// TIA Portal V20 program export: 1 tag tables, 2 data types, 6 data blocks, 9 code blocks (in call order from the OBs), 0 instance data blocks

VAR_GLOBAL   // PLC tag table "Default tag table"
   OpenCmd AT %M0.0 : Bool;
   CloseCmd AT %M0.1 : Bool;
   OpenFB AT %M0.2 : Bool;
   ClosedFB AT %M0.3 : Bool;
   LocalMode AT %M0.4 : Bool;
   Healthy AT %M0.5 : Bool;
   OpenValve AT %M0.6 : Bool;
   CloseValve AT %M0.7 : Bool;
   Tag__639217692550262421 AT %I2.0 : Bool;
   Tag__639217692553776870 AT %I2.1 : Bool;
   Tag__639217692553954872 AT %I2.2 : Bool;
   Tag__639217692553954873 AT %I2.3 : Bool;
   Tag__639217692554216438 AT %I2.4 : Bool;
   Tag__639217692554394622 AT %I2.5 : Bool;
   Tag__639217692554432300 AT %I2.6 : Bool;
   Tag__639217692556336031 AT %I2.7 : Bool;
   Tag__639217692556550149 AT %I3.0 : Bool;
   Tag__639217692556680608 AT %I3.1 : Bool;
   Tag__639217692556821735 AT %I3.2 : Bool;
   Tag__639217692556891742 AT %I3.3 : Bool;
   Tag__639217692557049682 AT %I3.4 : Bool;
   Tag__639217692557209508 AT %I3.5 : Bool;
   Tag__639217692557209509 AT %I3.6 : Bool;
   Tag__639217692557471753 AT %I3.7 : Bool;
   Tag__639217692557529414 AT %I4.0 : Bool;
   Tag__639217692557689863 AT %I4.1 : Bool;
   Tag__639217692557850060 AT %I4.2 : Bool;
   Tag__639217692558010331 AT %I4.3 : Bool;
   Tag__639217692558171799 AT %I4.4 : Bool;
   Tag__639217692558331401 AT %I4.5 : Bool;
   Tag__639217692558488410 AT %I4.6 : Bool;
   Tag__639217692558802162 AT %I4.7 : Bool;
   Tag__639217692558961456 AT %I5.0 : Bool;
   Tag__639217692558971616 AT %I5.1 : Bool;
   Tag__639217692559129482 AT %I5.2 : Bool;
   Tag__639217692559281543 AT %I5.3 : Bool;
   Tag__639217692559443162 AT %I5.4 : Bool;
   Tag__639217692559601745 AT %I5.5 : Bool;
   Tag__639217692559760896 AT %I5.6 : Bool;
   Tag__639217692559921432 AT %I5.7 : Bool;
   Tag__639217692559921433 AT %I6.0 : Bool;
   Tag__639217692560082018 AT %I6.1 : Bool;
   Tag__639217692560402934 AT %I6.2 : Bool;
   Tag__639217692560402935 AT %I6.3 : Bool;
   Tag__639217692560583987 AT %I6.4 : Bool;
   Tag__639217692560723706 AT %I6.5 : Bool;
   Tag__639217692560880740 AT %I6.6 : Bool;
   Tag__639217692561041807 AT %I6.7 : Bool;
   Tag__639217692561206457 AT %I7.0 : Bool;
   Tag__639217692561359218 AT %I7.1 : Bool;
   Tag__639217692561520184 AT %I7.2 : Bool;
   Tag__639217692561520185 AT %I7.3 : Bool;
   Tag__639217692561802187 AT %I7.4 : Bool;
   Tag__639217692561935087 AT %I7.5 : Bool;
   Tag__639217692562065024 AT %I7.6 : Bool;
   Tag__639217692562223286 AT %I7.7 : Bool;
   Tag__639217692562383723 AT %I8.0 : Bool;
   Tag__639217692562543936 AT %I8.1 : Bool;
   Tag__639217692562543937 AT %I8.2 : Bool;
   Tag__639217692562862407 AT %I8.3 : Bool;
   Tag__639217692562862408 AT %I8.4 : Bool;
   Tag__639217692563093001 AT %I8.5 : Bool;
   Tag__639217692563182212 AT %I8.6 : Bool;
   Tag__639217692563343596 AT %I8.7 : Bool;
   Tag__639217692563511187 AT %I9.0 : Bool;
   Tag__639217692563662093 AT %I9.1 : Bool;
   Tag__639217692563662094 AT %I9.2 : Bool;
   Tag__639217692563823907 AT %I9.3 : Bool;
   Tag__639217692566083593 AT %I9.4 : Bool;
   Tag__639217692566201557 AT %I9.5 : Bool;
   Tag__639217692566360040 AT %I9.6 : Bool;
   Tag__639217692566517145 AT %I9.7 : Bool;
   Tag__639217692566674032 AT %I10.0 : Bool;
   Tag__639217692566832496 AT %I10.1 : Bool;
   Tag__639217692566832497 AT %I10.2 : Bool;
   Tag__639217692567184922 AT %I10.3 : Bool;
   Tag__639217692567336780 AT %I10.4 : Bool;
   Tag__639217692567388945 AT %I10.5 : Bool;
   Tag__639217692567546587 AT %I10.6 : Bool;
   Tag__639217692567707146 AT %I10.7 : Bool;
   Tag__639217692567868007 AT %I11.0 : Bool;
   Tag__639217692567868008 AT %I11.1 : Bool;
   Tag__639217692568025035 AT %I11.2 : Bool;
   Tag__639217692568182907 AT %I11.3 : Bool;
   Tag__639217692568341074 AT %I11.4 : Bool;
   Tag__639217692568550097 AT %I11.5 : Bool;
   Tag__639217692568683019 AT %I11.6 : Bool;
   Tag__639217692568840948 AT %I11.7 : Bool;
   Tag__639217692568971320 AT %I12.0 : Bool;
   Tag__639217692569119475 AT %I12.1 : Bool;
   Tag__639217692569298523 AT %I12.2 : Bool;
   Tag__639217692569460008 AT %I12.3 : Bool;
   Tag__639217692569619373 AT %I12.4 : Bool;
   Tag__639217692569780777 AT %I12.5 : Bool;
   Tag__639217692569780778 AT %I12.6 : Bool;
   Tag__639217692569942097 AT %I12.7 : Bool;
   Tag__639217692570102018 AT %I13.0 : Bool;
   Tag__639217692570262026 AT %I13.1 : Bool;
   Tag__639217692570422186 AT %I13.2 : Bool;
   Tag__639217692570422187 AT %I13.3 : Bool;
   Tag__639217692570583489 AT %I13.4 : Bool;
   Tag__639217692570745102 AT %I13.5 : Bool;
   Tag__639217692570906074 AT %I13.6 : Bool;
   Tag__639217692570906075 AT %I13.7 : Bool;
   Tag__639217692571063660 AT %I14.0 : Bool;
   Tag__639217692571223097 AT %I14.1 : Bool;
   Tag__639217692571384739 AT %I14.2 : Bool;
   Tag__639217692571544096 AT %I14.3 : Bool;
   Tag__639217692571703825 AT %I14.4 : Bool;
   Tag__639217692571865026 AT %I14.5 : Bool;
   Tag__639217692572024808 AT %I14.6 : Bool;
   Tag__639217692572184903 AT %I14.7 : Bool;
   Tag__639217692572395679 AT %I15.0 : Bool;
   Tag__639217692572536054 AT %I15.1 : Bool;
   Tag__639217692572670856 AT %I15.2 : Bool;
   Tag__639217692572707880 AT %I15.3 : Bool;
   Tag__639217692572861963 AT %I15.4 : Bool;
   Tag__639217692573067363 AT %I15.5 : Bool;
   Tag__639217692573180541 AT %I15.6 : Bool;
   Tag__639217692573357884 AT %I15.7 : Bool;
   Tag__639217692573503474 AT %I16.0 : Bool;
   Tag__639217692573503475 AT %I16.1 : Bool;
   Tag__639217692573691090 AT %I16.2 : Bool;
   Tag__639217692573812370 AT %I16.3 : Bool;
   Tag__639217692573973083 AT %I16.4 : Bool;
   Tag__639217692574133186 AT %I16.5 : Bool;
   Tag__639217692574289638 AT %I16.6 : Bool;
   Tag__639217692574448526 AT %I16.7 : Bool;
   Tag__639217692574609334 AT %I17.0 : Bool;
   Tag__639217692574768434 AT %I17.1 : Bool;
   Tag__639217692574930294 AT %I17.2 : Bool;
   Tag__639217692575083184 AT %I17.3 : Bool;
   Tag__639217692575261129 AT %I17.4 : Bool;
   Tag__639217692575419042 AT %I17.5 : Bool;
   Tag__639217692575539382 AT %I17.6 : Bool;
   Tag__639217692575911602 AT %I17.7 : Bool;
   Tag__639217692576029509 AT %I18.0 : Bool;
   Tag__639217692576029510 AT %I18.1 : Bool;
   Tag__639217692576190207 AT %I18.2 : Bool;
   Tag__639217692576351259 AT %I18.3 : Bool;
   Tag__639217692576511022 AT %I18.4 : Bool;
   Tag__639217692576672087 AT %I18.5 : Bool;
   Tag__639217692576832345 AT %I18.6 : Bool;
   Tag__639217692576952866 AT %I18.7 : Bool;
   Tag__639217692576990475 AT %I19.0 : Bool;
   Tag__639217692577151896 AT %I19.1 : Bool;
   Tag__639217692577372028 AT %I19.2 : Bool;
   Tag__639217692577469814 AT %I19.3 : Bool;
   Tag__639217692577766896 AT %I19.4 : Bool;
   Tag__639217692577926746 AT %I19.5 : Bool;
   Tag__639217692578046402 AT %I19.6 : Bool;
   Tag__639217692578046403 AT %I19.7 : Bool;
   Tag__639217692578204423 AT %I20.0 : Bool;
   Tag__639217692578364346 AT %I20.1 : Bool;
   Tag__639217692578525327 AT %I20.2 : Bool;
   Tag__639217692578706091 AT %I20.3 : Bool;
   Tag__639217692578841403 AT %I20.4 : Bool;
   Tag__639217692579004858 AT %I20.5 : Bool;
   Tag__639217692579155731 AT %I20.6 : Bool;
   Tag__639217692579314254 AT %I20.7 : Bool;
   Tag__639217692579314255 AT %I21.0 : Bool;
   Tag__639217692579474584 AT %I21.1 : Bool;
   Tag__639217692579635203 AT %I21.2 : Bool;
   Tag__639217692579794995 AT %I21.3 : Bool;
   Tag__639217692579955090 AT %I21.4 : Bool;
   Tag__639217692580275677 AT %I21.5 : Bool;
   Tag__639217692580432274 AT %I21.6 : Bool;
   Tag__639217692580552766 AT %I21.7 : Bool;
   Tag__639217692580590363 AT %I22.0 : Bool;
   Tag__639217692580751532 AT %I22.1 : Bool;
   Tag__639217692580913166 AT %I22.2 : Bool;
   Tag__639217692581133835 AT %I22.3 : Bool;
   Tag__639217692581227406 AT %I22.4 : Bool;
   Tag__639217692581387294 AT %I22.5 : Bool;
   Tag__639217692581507780 AT %I22.6 : Bool;
   Tag__639217692581545371 AT %I22.7 : Bool;
   Tag__639217692581704532 AT %I23.0 : Bool;
   Tag__639217692581863905 AT %I23.1 : Bool;
   Tag__639217692581863906 AT %I23.2 : Bool;
   Tag__639217692582023588 AT %I23.3 : Bool;
   Tag__639217692582184822 AT %I23.4 : Bool;
   Tag__639217692582344335 AT %I23.5 : Bool;
   Tag__639217692582505209 AT %I23.6 : Bool;
   Tag__639217692582505210 AT %I23.7 : Bool;
   Tag__639217692582664098 AT %I24.0 : Bool;
   Tag__639217692582825326 AT %I24.1 : Bool;
   Tag__639217692582994863 AT %I24.2 : Bool;
   Tag__639217692583198482 AT %I24.3 : Bool;
   Tag__639217692583329182 AT %I24.4 : Bool;
   Tag__639217692583430354 AT %I24.5 : Bool;
   Tag__639217692583542618 AT %I24.6 : Bool;
   Tag__639217692583692939 AT %I24.7 : Bool;
   Tag__639217692585720764 AT %I25.0 : Bool;
   Tag__639217692585760931 AT %I25.1 : Bool;
   Tag__639217692585920591 AT %I25.2 : Bool;
   Tag__639217692586101165 AT %I25.3 : Bool;
   Tag__639217692586241395 AT %I25.4 : Bool;
   Tag__639217692586241396 AT %I25.5 : Bool;
   Tag__639217692586401865 AT %I25.6 : Bool;
   Tag__639217692586559348 AT %I25.7 : Bool;
   Tag__639217692586717642 AT %I26.0 : Bool;
   Tag__639217692586876705 AT %I26.1 : Bool;
   Tag__639217692587037050 AT %I26.2 : Bool;
   Tag__639217692587198156 AT %I26.3 : Bool;
   Tag__639217692587198157 AT %I26.4 : Bool;
   Tag__639217692587438593 AT %I26.5 : Bool;
   Tag__639217692587516326 AT %I26.6 : Bool;
   Tag__639217692587676973 AT %I26.7 : Bool;
   Tag__639217692587676974 AT %I27.0 : Bool;
   Tag__639217692587854158 AT %I27.1 : Bool;
   Tag__639217692587995295 AT %I27.2 : Bool;
   Tag__639217692588156000 AT %I27.3 : Bool;
   Tag__639217692588379878 AT %I27.4 : Bool;
   Tag__639217692588550268 AT %I27.5 : Bool;
   Tag__639217692588708101 AT %I27.6 : Bool;
   Tag__639217692588866833 AT %I27.7 : Bool;
   Tag__639217692589023179 AT %I28.0 : Bool;
   Tag__639217692589158483 AT %I28.1 : Bool;
   Tag__639217692589208458 AT %I28.2 : Bool;
   Tag__639217692589366891 AT %I28.3 : Bool;
   Tag__639217692589526977 AT %I28.4 : Bool;
   Tag__639217692589687241 AT %I28.5 : Bool;
   Tag__639217692589848658 AT %I28.6 : Bool;
   Tag__639217692589848659 AT %I28.7 : Bool;
   Tag__639217692590010039 AT %I29.0 : Bool;
   Tag__639217692590170658 AT %I29.1 : Bool;
   Tag__639217692590328833 AT %I29.2 : Bool;
   Tag__639217692590485955 AT %I29.3 : Bool;
   Tag__639217692590485956 AT %I29.4 : Bool;
   Tag__639217692590645258 AT %I29.5 : Bool;
   Tag__639217692590805752 AT %I29.6 : Bool;
   Tag__639217692590966425 AT %I29.7 : Bool;
   Tag__639217692590966426 AT %I30.0 : Bool;
   Tag__639217692591127321 AT %I30.1 : Bool;
   Tag__639217692591285391 AT %I30.2 : Bool;
   Tag__639217692591446446 AT %I30.3 : Bool;
   Tag__639217692591605376 AT %I30.4 : Bool;
   Tag__639217692591923527 AT %I30.5 : Bool;
   Tag__639217692591923528 AT %I30.6 : Bool;
   Tag__639217692592084854 AT %I30.7 : Bool;
   Tag__639217692592246014 AT %I31.0 : Bool;
   Tag__639217692592406057 AT %I31.1 : Bool;
   Tag__639217692592406058 AT %I31.2 : Bool;
   Tag__639217692592567050 AT %I31.3 : Bool;
   Tag__639217692592727547 AT %I31.4 : Bool;
   Tag__639217692592888082 AT %I31.5 : Bool;
   Tag__639217692593114463 AT %I31.6 : Bool;
   Tag__639217692593206619 AT %I31.7 : Bool;
   Tag__639217692593364125 AT %I32.0 : Bool;
   Tag__639217692593535630 AT %I32.1 : Bool;
   Tag__639217692593656106 AT %I32.2 : Bool;
   Tag__639217692593702147 AT %I32.3 : Bool;
   Tag__639217692593935520 AT %I32.4 : Bool;
   Tag__639217692594074769 AT %I32.5 : Bool;
   Tag__639217692594204786 AT %I32.6 : Bool;
   Tag__639217692594204787 AT %I32.7 : Bool;
   Tag__639217692594365259 AT %I33.0 : Bool;
   Tag__639217692594522265 AT %I33.1 : Bool;
   Tag__639217692594681744 AT %I33.2 : Bool;
   Tag__639217692594681745 AT %I33.3 : Bool;
   Tag__639217692594842324 AT %I33.4 : Bool;
   Tag__639217692595003601 AT %I33.5 : Bool;
   Tag__639217692595162932 AT %I33.6 : Bool;
   Tag__639217692595295217 AT %I33.7 : Bool;
   Tag__639217692595321829 AT %I34.0 : Bool;
   Tag__639217692595479808 AT %I34.1 : Bool;
   Tag__639217692595637197 AT %I34.2 : Bool;
   Tag__639217692595797438 AT %I34.3 : Bool;
   Tag__639217692595959028 AT %I34.4 : Bool;
   Tag__639217692596136048 AT %I34.5 : Bool;
   Tag__639217692596337735 AT %I34.6 : Bool;
   Tag__639217692596435546 AT %I34.7 : Bool;
   Tag__639217692596435547 AT %I35.0 : Bool;
   Tag__639217692596596639 AT %I35.1 : Bool;
   Tag__639217692596754611 AT %I35.2 : Bool;
   Tag__639217692596914545 AT %I35.3 : Bool;
   Tag__639217692597075234 AT %I35.4 : Bool;
   Tag__639217692597075235 AT %I35.5 : Bool;
   Tag__639217692597235934 AT %I35.6 : Bool;
   Tag__639217692597397011 AT %I35.7 : Bool;
   Tag__639217692597554180 AT %I36.0 : Bool;
   Tag__639217692597711217 AT %I36.1 : Bool;
   Tag__639217692597871107 AT %I36.2 : Bool;
   Tag__639217692598028494 AT %I36.3 : Bool;
   Tag__639217692598185471 AT %I36.4 : Bool;
   Tag__639217692598185472 AT %I36.5 : Bool;
   Tag__639217692598345589 AT %I36.6 : Bool;
   Tag__639217692598572817 AT %I36.7 : Bool;
   Tag__639217692598703247 AT %I37.0 : Bool;
   Tag__639217692598865809 AT %I37.1 : Bool;
   Tag__639217692599003448 AT %I37.2 : Bool;
   Tag__639217692599080153 AT %I37.3 : Bool;
   Tag__639217692599295021 AT %I37.4 : Bool;
   Tag__639217692599434105 AT %I37.5 : Bool;
   Tag__639217692599574585 AT %I37.6 : Bool;
   Tag__639217692599692113 AT %I37.7 : Bool;
   Tag__639217692599852177 AT %I38.0 : Bool;
   Tag__639217692599852178 AT %I38.1 : Bool;
   Tag__639217692600013096 AT %I38.2 : Bool;
   Tag__639217692600225652 AT %I38.3 : Bool;
   Tag__639217692600329437 AT %I38.4 : Bool;
   Tag__639217692600517312 AT %I38.5 : Bool;
   Tag__639217692600648060 AT %I38.6 : Bool;
   Tag__639217692600809555 AT %I38.7 : Bool;
   Tag__639217692600970188 AT %I39.0 : Bool;
   Tag__639217692600970189 AT %I39.1 : Bool;
   Tag__639217692601290117 AT %I39.2 : Bool;
   Tag__639217692601576181 AT %I39.3 : Bool;
   Tag__639217692601764420 AT %I39.4 : Bool;
   Tag__639217692601904130 AT %I39.5 : Bool;
   Tag__639217692601921632 AT %I39.6 : Bool;
   Tag__639217692602082038 AT %I39.7 : Bool;
   Tag__639217692602243355 AT %I40.0 : Bool;
   Tag__639217692602403696 AT %I40.1 : Bool;
   Tag__639217692602403697 AT %I40.2 : Bool;
   Tag__639217692602561458 AT %I40.3 : Bool;
   Tag__639217692602720965 AT %I40.4 : Bool;
   Tag__639217692602881697 AT %I40.5 : Bool;
   Tag__639217692602881698 AT %I40.6 : Bool;
   Tag__639217692603041227 AT %I40.7 : Bool;
   Tag__639217692603201062 AT %I41.0 : Bool;
   Tag__639217692603432857 AT %I41.1 : Bool;
   Tag__639217692603526128 AT %I41.2 : Bool;
   Tag__639217692603677627 AT %I41.3 : Bool;
   Tag__639217692603839177 AT %I41.4 : Bool;
   Tag__639217692603998759 AT %I41.5 : Bool;
   Tag__639217692603998760 AT %I41.6 : Bool;
   Tag__639217692604301271 AT %I41.7 : Bool;
   Tag__639217692604446823 AT %I42.0 : Bool;
   Tag__639217692604524554 AT %I42.1 : Bool;
   Tag__639217692604674613 AT %I42.2 : Bool;
   Tag__639217692604834416 AT %I42.3 : Bool;
   Tag__639217692605944492 AT %I42.4 : Bool;
   Tag__639217692606105425 AT %I42.5 : Bool;
   Tag__639217692606105426 AT %I42.6 : Bool;
   Tag__639217692606285541 AT %I42.7 : Bool;
   Tag__639217692606426194 AT %I43.0 : Bool;
   Tag__639217692606584564 AT %I43.1 : Bool;
   Tag__639217692606742338 AT %I43.2 : Bool;
   Tag__639217692606904136 AT %I43.3 : Bool;
   Tag__639217692607062435 AT %I43.4 : Bool;
   Tag__639217692607224125 AT %I43.5 : Bool;
   Tag__639217692607224126 AT %I43.6 : Bool;
   Tag__639217692607485341 AT %I43.7 : Bool;
   Tag__639217692607543000 AT %I44.0 : Bool;
   Tag__639217692607763945 AT %I44.1 : Bool;
   Tag__639217692607861770 AT %I44.2 : Bool;
   Tag__639217692608018680 AT %I44.3 : Bool;
   Tag__639217692608018681 AT %I44.4 : Bool;
   Tag__639217692608238678 AT %I44.5 : Bool;
   Tag__639217692608335365 AT %I44.6 : Bool;
   Tag__639217692608493637 AT %I44.7 : Bool;
   Tag__639217692608653174 AT %I45.0 : Bool;
   Tag__639217692608812275 AT %I45.1 : Bool;
   Tag__639217692608812276 AT %I45.2 : Bool;
   Tag__639217692609128733 AT %I45.3 : Bool;
   Tag__639217692609128734 AT %I45.4 : Bool;
   Tag__639217692609289890 AT %I45.5 : Bool;
   Tag__639217692609532283 AT %I45.6 : Bool;
   Tag__639217692609702548 AT %I45.7 : Bool;
   Tag__639217692609862538 AT %I46.0 : Bool;
   Tag__639217692609862539 AT %I46.1 : Bool;
   Tag__639217692610182631 AT %I46.2 : Bool;
   Tag__639217692610182632 AT %I46.3 : Bool;
   Tag__639217692610403611 AT %I46.4 : Bool;
   Tag__639217692610501805 AT %I46.5 : Bool;
   Tag__639217692610661275 AT %I46.6 : Bool;
   Tag__639217692610661276 AT %I46.7 : Bool;
   Tag__639217692610983046 AT %I47.0 : Bool;
   Tag__639217692610983047 AT %I47.1 : Bool;
   Tag__639217692611192346 AT %I47.2 : Bool;
   Tag__639217692611310653 AT %I47.3 : Bool;
   Tag__639217692611461334 AT %I47.4 : Bool;
   Tag__639217692611622448 AT %I47.5 : Bool;
   Tag__639217692611781748 AT %I47.6 : Bool;
   Tag__639217692611781749 AT %I47.7 : Bool;
   Tag__639217692612263475 AT %Q2.0 : Bool;
   Tag__639217692612423650 AT %Q2.1 : Bool;
   Tag__639217692612585355 AT %Q2.2 : Bool;
   Tag__639217692612746418 AT %Q2.3 : Bool;
   Tag__639217692612905975 AT %Q2.4 : Bool;
   Tag__639217692612905976 AT %Q2.5 : Bool;
   Tag__639217692613224334 AT %Q2.6 : Bool;
   Tag__639217692613431048 AT %Q2.7 : Bool;
   Tag__639217692613549459 AT %Q3.0 : Bool;
   Tag__639217692613549460 AT %Q3.1 : Bool;
   Tag__639217692613700358 AT %Q3.2 : Bool;
   Tag__639217692613860481 AT %Q3.3 : Bool;
   Tag__639217692614018559 AT %Q3.4 : Bool;
   Tag__639217692614298000 AT %Q3.5 : Bool;
   Tag__639217692614480374 AT %Q3.6 : Bool;
   Tag__639217692614684823 AT %Q3.7 : Bool;
   Tag__639217692614993876 AT %Q4.0 : Bool;
   Tag__639217692615192661 AT %Q4.1 : Bool;
   Tag__639217692615372374 AT %Q4.2 : Bool;
   Tag__639217692615821386 AT %Q4.3 : Bool;
   Tag__639217692615982422 AT %Q4.4 : Bool;
   Tag__639217692616141851 AT %Q4.5 : Bool;
   Tag__639217692616362637 AT %Q4.6 : Bool;
   Tag__639217692616460481 AT %Q4.7 : Bool;
   Tag__639217692616782087 AT %Q5.0 : Bool;
   Tag__639217692616782088 AT %Q5.1 : Bool;
   Tag__639217692616940617 AT %Q5.2 : Bool;
   Tag__639217692617097153 AT %Q5.3 : Bool;
   Tag__639217692617257965 AT %Q5.4 : Bool;
   Tag__639217692617425635 AT %Q5.5 : Bool;
   Tag__639217692617581306 AT %Q5.6 : Bool;
   Tag__639217692617739154 AT %Q5.7 : Bool;
   Tag__639217692617899719 AT %Q6.0 : Bool;
   Tag__639217692618058569 AT %Q6.1 : Bool;
   Tag__639217692618215933 AT %Q6.2 : Bool;
   Tag__639217692618373391 AT %Q6.3 : Bool;
   Tag__639217692618554770 AT %Q6.4 : Bool;
   Tag__639217692618760680 AT %Q6.5 : Bool;
   Tag__639217692618931105 AT %Q6.6 : Bool;
   Tag__639217692619091004 AT %Q6.7 : Bool;
   Tag__639217692619165425 AT %Q7.0 : Bool;
   Tag__639217692619325369 AT %Q7.1 : Bool;
   Tag__639217692619487118 AT %Q7.2 : Bool;
   Tag__639217692619487119 AT %Q7.3 : Bool;
   Tag__639217692619648292 AT %Q7.4 : Bool;
   Tag__639217692619808948 AT %Q7.5 : Bool;
   Tag__639217692620036810 AT %Q7.6 : Bool;
   Tag__639217692620197299 AT %Q7.7 : Bool;
   Tag__639217692620337293 AT %Q8.0 : Bool;
   Tag__639217692620357294 AT %Q8.1 : Bool;
   Tag__639217692620515379 AT %Q8.2 : Bool;
   Tag__639217692620675332 AT %Q8.3 : Bool;
   Tag__639217692620835634 AT %Q8.4 : Bool;
   Tag__639217692620992973 AT %Q8.5 : Bool;
   Tag__639217692621152065 AT %Q8.6 : Bool;
   Tag__639217692621309565 AT %Q8.7 : Bool;
   Tag__639217692621469714 AT %Q9.0 : Bool;
   Tag__639217692621469715 AT %Q9.1 : Bool;
   Tag__639217692621630499 AT %Q9.2 : Bool;
   Tag__639217692621906549 AT %Q9.3 : Bool;
   Tag__639217692621950360 AT %Q9.4 : Bool;
   Tag__639217692622111179 AT %Q9.5 : Bool;
   Tag__639217692622292619 AT %Q9.6 : Bool;
   Tag__639217692622426875 AT %Q9.7 : Bool;
   Tag__639217692622426876 AT %Q10.0 : Bool;
   Tag__639217692622587394 AT %Q10.1 : Bool;
   Tag__639217692622746975 AT %Q10.2 : Bool;
   Tag__639217692622906735 AT %Q10.3 : Bool;
   Tag__639217692623064209 AT %Q10.4 : Bool;
   Tag__639217692623222595 AT %Q10.5 : Bool;
   Tag__639217692623222596 AT %Q10.6 : Bool;
   Tag__639217692623428677 AT %Q10.7 : Bool;
   Tag__639217692623552568 AT %Q11.0 : Bool;
   Tag__639217692623706024 AT %Q11.1 : Bool;
   Tag__639217692623866625 AT %Q11.2 : Bool;
   Tag__639217692624026402 AT %Q11.3 : Bool;
   Tag__639217692624188100 AT %Q11.4 : Bool;
   Tag__639217692624296413 AT %Q11.5 : Bool;
   Tag__639217692624349590 AT %Q11.6 : Bool;
   Tag__639217692624607979 AT %Q11.7 : Bool;
   Tag__639217692624665644 AT %Q12.0 : Bool;
   Tag__639217692624979691 AT %Q12.1 : Bool;
   Tag__639217692625112094 AT %Q12.2 : Bool;
   Tag__639217692625921588 AT %Q12.3 : Bool;
   Tag__639217692626087431 AT %Q12.4 : Bool;
   Tag__639217692626253351 AT %Q12.5 : Bool;
   Tag__639217692626352897 AT %Q12.6 : Bool;
   Tag__639217692626510009 AT %Q12.7 : Bool;
   Tag__639217692626671657 AT %Q13.0 : Bool;
   Tag__639217692626671658 AT %Q13.1 : Bool;
   Tag__639217692626833520 AT %Q13.2 : Bool;
   Tag__639217692626994806 AT %Q13.3 : Bool;
   Tag__639217692627254988 AT %Q13.4 : Bool;
   Tag__639217692627312671 AT %Q13.5 : Bool;
   Tag__639217692627473354 AT %Q13.6 : Bool;
   Tag__639217692627673115 AT %Q13.7 : Bool;
   Tag__639217692627811109 AT %Q14.0 : Bool;
   Tag__639217692627949093 AT %Q14.1 : Bool;
   Tag__639217692628089666 AT %Q14.2 : Bool;
   Tag__639217692628107166 AT %Q14.3 : Bool;
   Tag__639217692628336120 AT %Q14.4 : Bool;
   Tag__639217692628492917 AT %Q14.5 : Bool;
   Tag__639217692628623290 AT %Q14.6 : Bool;
   Tag__639217692628761042 AT %Q14.7 : Bool;
   Tag__639217692628899816 AT %Q15.0 : Bool;
   Tag__639217692628972569 AT %Q15.1 : Bool;
   Tag__639217692629072663 AT %Q15.2 : Bool;
   Tag__639217692629316047 AT %Q15.3 : Bool;
   Tag__639217692629373725 AT %Q15.4 : Bool;
   Tag__639217692629533777 AT %Q15.5 : Bool;
   Tag__639217692629693574 AT %Q15.6 : Bool;
   Tag__639217692629851555 AT %Q15.7 : Bool;
   Tag__639217692630008442 AT %Q16.0 : Bool;
   Tag__639217692630168713 AT %Q16.1 : Bool;
   Tag__639217692630329520 AT %Q16.2 : Bool;
   Tag__639217692630490637 AT %Q16.3 : Bool;
   Tag__639217692630661059 AT %Q16.4 : Bool;
   Tag__639217692630807879 AT %Q16.5 : Bool;
   Tag__639217692630939597 AT %Q16.6 : Bool;
   Tag__639217692631073684 AT %Q16.7 : Bool;
   Tag__639217692631183654 AT %Q17.0 : Bool;
   Tag__639217692631183655 AT %Q17.1 : Bool;
   Tag__639217692631342517 AT %Q17.2 : Bool;
   Tag__639217692631504108 AT %Q17.3 : Bool;
   Tag__639217692631664286 AT %Q17.4 : Bool;
   Tag__639217692631824426 AT %Q17.5 : Bool;
   Tag__639217692631981364 AT %Q17.6 : Bool;
   Tag__639217692631981365 AT %Q17.7 : Bool;
   Tag__639217692632142556 AT %Q18.0 : Bool;
   Tag__639217692632301255 AT %Q18.1 : Bool;
   Tag__639217692632461403 AT %Q18.2 : Bool;
   Tag__639217692632622376 AT %Q18.3 : Bool;
   Tag__639217692632622377 AT %Q18.4 : Bool;
   Tag__639217692632781836 AT %Q18.5 : Bool;
   Tag__639217692633119556 AT %Q18.6 : Bool;
   Tag__639217692633257667 AT %Q18.7 : Bool;
   Tag__639217692633257668 AT %Q19.0 : Bool;
   Tag__639217692633606974 AT %Q19.1 : Bool;
   Tag__639217692633797544 AT %Q19.2 : Bool;
   Tag__639217692633935297 AT %Q19.3 : Bool;
   Tag__639217692634052982 AT %Q19.4 : Bool;
   Tag__639217692634250953 AT %Q19.5 : Bool;
   Tag__639217692634367505 AT %Q19.6 : Bool;
   Tag__639217692634526933 AT %Q19.7 : Bool;
   Tag__639217692634686575 AT %Q20.0 : Bool;
   Tag__639217692634847392 AT %Q20.1 : Bool;
   Tag__639217692635084699 AT %Q20.2 : Bool;
   Tag__639217692635166263 AT %Q20.3 : Bool;
   Tag__639217692635324026 AT %Q20.4 : Bool;
   Tag__639217692635482506 AT %Q20.5 : Bool;
   Tag__639217692635482507 AT %Q20.6 : Bool;
   Tag__639217692635642498 AT %Q20.7 : Bool;
   Tag__639217692635802017 AT %Q21.0 : Bool;
   Tag__639217692636027800 AT %Q21.1 : Bool;
   Tag__639217692636167857 AT %Q21.2 : Bool;
   Tag__639217692636298889 AT %Q21.3 : Bool;
   Tag__639217692636348888 AT %Q21.4 : Bool;
   Tag__639217692636549597 AT %Q21.5 : Bool;
   Tag__639217692636666551 AT %Q21.6 : Bool;
   Tag__639217692636827995 AT %Q21.7 : Bool;
   Tag__639217692636988786 AT %Q22.0 : Bool;
   Tag__639217692636988787 AT %Q22.1 : Bool;
   Tag__639217692637150621 AT %Q22.2 : Bool;
   Tag__639217692637311136 AT %Q22.3 : Bool;
   Tag__639217692637471435 AT %Q22.4 : Bool;
   Tag__639217692637631790 AT %Q22.5 : Bool;
   Tag__639217692637789494 AT %Q22.6 : Bool;
   Tag__639217692637950184 AT %Q22.7 : Bool;
   Tag__639217692637950185 AT %Q23.0 : Bool;
   Tag__639217692638109462 AT %Q23.1 : Bool;
   Tag__639217692638276714 AT %Q23.2 : Bool;
   Tag__639217692638427229 AT %Q23.3 : Bool;
   Tag__639217692638586533 AT %Q23.4 : Bool;
   Tag__639217692638747466 AT %Q23.5 : Bool;
   Tag__639217692638904386 AT %Q23.6 : Bool;
   Tag__639217692639063833 AT %Q23.7 : Bool;
   Tag__639217692639078981 AT %Q24.0 : Bool;
   Tag__639217692639243768 AT %Q24.1 : Bool;
   Tag__639217692639383298 AT %Q24.2 : Bool;
   Tag__639217692639542163 AT %Q24.3 : Bool;
   Tag__639217692639701541 AT %Q24.4 : Bool;
   Tag__639217692639892825 AT %Q24.5 : Bool;
   Tag__639217692640016631 AT %Q24.6 : Bool;
   Tag__639217692640016632 AT %Q24.7 : Bool;
   Tag__639217692640175734 AT %Q25.0 : Bool;
   Tag__639217692640332797 AT %Q25.1 : Bool;
   Tag__639217692640492541 AT %Q25.2 : Bool;
   Tag__639217692640652754 AT %Q25.3 : Bool;
   Tag__639217692640652755 AT %Q25.4 : Bool;
   Tag__639217692640812694 AT %Q25.5 : Bool;
   Tag__639217692640972759 AT %Q25.6 : Bool;
   Tag__639217692641133541 AT %Q25.7 : Bool;
   Tag__639217692641370581 AT %Q26.0 : Bool;
   Tag__639217692641539941 AT %Q26.1 : Bool;
   Tag__639217692641669868 AT %Q26.2 : Bool;
   Tag__639217692641679864 AT %Q26.3 : Bool;
   Tag__639217692641838308 AT %Q26.4 : Bool;
   Tag__639217692641998720 AT %Q26.5 : Bool;
   Tag__639217692642156578 AT %Q26.6 : Bool;
   Tag__639217692642313321 AT %Q26.7 : Bool;
   Tag__639217692642472571 AT %Q27.0 : Bool;
   Tag__639217692642631876 AT %Q27.1 : Bool;
   Tag__639217692642631877 AT %Q27.2 : Bool;
   Tag__639217692642792640 AT %Q27.3 : Bool;
   Tag__639217692642950472 AT %Q27.4 : Bool;
   Tag__639217692643191744 AT %Q27.5 : Bool;
   Tag__639217692643266837 AT %Q27.6 : Bool;
   Tag__639217692643431479 AT %Q27.7 : Bool;
END_VAR

TYPE "UDT_Valve_Config"
// Per-valve physical channel assignment. 0 = unassigned (valve runs on symbolic simulation). A nonzero value is an index into IO_Buffer_DB.DI[]/DQ[] - our own abstract channel numbering, translated to real hardware addresses in one place only (see FC_IoMapper).
// stored: IsFailsafeCompliant false
   STRUCT
      OpenFb_Channel : Int;
      ClosedFb_Channel : Int;
      Healthy_Channel : Int;
      LocalMode_Channel : Int;
      OpenCmd_Channel : Int;
      CloseCmd_Channel : Int;
   END_STRUCT;
END_TYPE

TYPE "Valve_IO"
// stored: IsFailsafeCompliant false
   STRUCT
      Configured : Bool;
      OpenCmd : Bool;
      CloseCmd : Bool;
      LocalMode : Bool;
      Healthy : Bool;
      OpenFB : Bool;
      ClosedFB : Bool;
      OpenValve : Bool;
      CloseValve : Bool;
      TimerOpen : TON_TIME;
      TimerClose : TON_TIME;
   END_STRUCT;
END_TYPE

DATA_BLOCK "Diag_DB"   // DB
{ S7_Optimized_Access := 'TRUE' }
VERSION : 0.1
// Station health, written by OB86 (RackOrStationFailure). Until this existed, an ET200SP could lose power and nothing in the system noticed: the valves on it simply stopped answering while the HMI carried on showing their last known positions as though they were live. Stale data presented as current is the actual hazard here, more than the loss of control - an operator plans a ballast transfer on positions that stopped being true ten minutes ago. The three hardware identifiers are data rather than code so that re-adding a station in TIA, which reassigns them, does not require an SCL edit. Read the current values off the SYSTEM DIAGNOSTICS screen: every device tile shows its identifier beneath the name.
// stored: AutoNumber true, IsOnlyStoredInLoadMemory false, IsRetainMemResEnabled false, IsWriteProtectedInAS false, MemoryReserve 100
   VAR
      Laddr_AFT : UInt := 273;   // Hardware identifier of ET200SP_AFT. Read off the SYSTEM DIAGNOSTICS screen - each device tile shows it under the name. Held here rather than in OB86 so that re-adding a station in TIA, which reassigns identifiers, is a data change and not a code change.
      Laddr_MID : UInt := 288;   // Hardware identifier of ET200SP_MID.
      Laddr_FWD : UInt := 306;   // Hardware identifier of ET200SP_FWD.
      AftLost : Bool;   // ET200SP_AFT is off the network. Valves 1-27 are unreachable and whatever the HMI shows for them is stale.
      MidLost : Bool;   // ET200SP_MID is off the network. Valves 28-54 are unreachable.
      FwdLost : Bool;   // ET200SP_FWD is off the network. Valves 55-89 are unreachable.
      UnknownLost : Bool;   // A station failed whose hardware identifier matches none of the three above. Means either the identifiers were reassigned and this DB was not updated, or a device exists that OB86 does not know about. Never silently ignored - that would hide a real station failure.
      AnyStationLost : Bool;   // Any of the four flags above. One bit for a screen to watch instead of ORing four.
      LastUnknownLaddr : UInt;   // The unrecognised identifier, kept so it can be looked up on the SYSTEM DIAGNOSTICS screen rather than guessed at.
      AftLossCount : Int;   // How many times AFT has dropped since startup. A station that is cleanly down reads 1; one that is flapping on a bad cable or a loose connector climbs, and that difference does not show in the status bit alone.
      MidLossCount : Int;   // Drop count for MID.
      FwdLossCount : Int;   // Drop count for FWD.
      ModuleFault : Bool;   // LATCHED: an I/O module raised a diagnostic. Cleared only by ModuleFaultAck - never self-clearing, see OB82.
      ModuleFaultAck : Bool;   // Write TRUE to clear ModuleFault. FB_ValveLoop consumes and clears this.
      ModuleEventCount : Int;   // Total OB82 events since CPU start. Rising with no new fault = a module chattering.
      LastModuleLaddr : UInt;   // Hardware identifier from the most recent OB82 event - identifies WHICH module.
      LastModuleIoState : Word;   // Raw IO_State word from the most recent OB82 event. Stored undecoded on purpose.
      LastModuleChannel : UInt;   // Channel number from the most recent OB82 event - narrows a fault to one terminal.
      LastModuleMultiError : Bool;   // TRUE if that event carried more than one error.
      NewModuleEvent : Bool;   // Set by OB82, consumed by FB_ValveLoop. The decode deliberately lives in FB_ValveLoop, not OB82, so it can be tested from a watch table - OB82 itself cannot be triggered in PLCSIM.
      ModuleLaddr : Array[1..36] of UInt;   // Hardware identifier of each I/O module, read from the PLC system constants 2026-09-10. Index order is RACK order: 1-11 AFT slots 1-11, 12-22 MID slots 1-11, 23-36 FWD slots 1-14. Held as DATA, not literals in SCL, for the same reason as Laddr_AFT/MID/FWD above. WARNING: re-adding a module in TIA reassigns these, and a shifted table would name the WRONG module - the unknown handler only catches a MISSING entry. Re-read the system constants after any hardware change. Note AFT is not contiguous (DQ ST_1 is 281, between the DI values) so a range check cannot substitute for this table.
      W_ModuleFault : Array[0..2] of Word;   // One LATCHED bit per I/O module. Module index i (1..36) is word (i-1)/16, bit (i-1) MOD 16 - the same packing the valve alarm words use. Cleared only by ModuleFaultAck.
      UnknownModuleFault : Bool;   // An OB82 event arrived whose LADDR is not in ModuleLaddr[]. Means the table is stale or an unexpected device reported. Never silently dropped.
      UnknownModuleLaddr : UInt;   // The unrecognised identifier, so a stale table can be diagnosed.
   END_VAR
BEGIN
   ModuleLaddr[1] := 280;
   ModuleLaddr[2] := 282;
   ModuleLaddr[3] := 283;
   ModuleLaddr[4] := 284;
   ModuleLaddr[5] := 285;
   ModuleLaddr[6] := 286;
   ModuleLaddr[7] := 287;
   ModuleLaddr[8] := 281;
   ModuleLaddr[9] := 270;
   ModuleLaddr[10] := 271;
   ModuleLaddr[11] := 272;
   ModuleLaddr[12] := 295;
   ModuleLaddr[13] := 296;
   ModuleLaddr[14] := 297;
   ModuleLaddr[15] := 298;
   ModuleLaddr[16] := 299;
   ModuleLaddr[17] := 300;
   ModuleLaddr[18] := 301;
   ModuleLaddr[19] := 302;
   ModuleLaddr[20] := 303;
   ModuleLaddr[21] := 304;
   ModuleLaddr[22] := 305;
   ModuleLaddr[23] := 313;
   ModuleLaddr[24] := 314;
   ModuleLaddr[25] := 315;
   ModuleLaddr[26] := 316;
   ModuleLaddr[27] := 317;
   ModuleLaddr[28] := 318;
   ModuleLaddr[29] := 319;
   ModuleLaddr[30] := 320;
   ModuleLaddr[31] := 321;
   ModuleLaddr[32] := 322;
   ModuleLaddr[33] := 323;
   ModuleLaddr[34] := 324;
   ModuleLaddr[35] := 325;
   ModuleLaddr[36] := 326;
END_DATA_BLOCK

DATA_BLOCK "Valve_Channels_DB"   // DB9
{ S7_Optimized_Access := 'TRUE' }
VERSION : 0.1
// Per-valve physical channel assignment, as six parallel flat arrays (one per UDT_Valve_Config field) rather than an array of the struct itself - Openness Import rejects StartValues on struct-typed array elements (confirmed via direct testing 2026-08-13, every encoding tried), while flat arrays of a simple type accept per-index StartValues cleanly, same as Valve_Meta_DB. Populated from the proposed station-by-zone channel assignment (AFT->ET200SP_AFT, ER->MID, FWD->FWD), reviewed and confirmed by the client before this import.
// stored: AutoNumber true, IsOnlyStoredInLoadMemory false, IsRetainMemResEnabled false, IsWriteProtectedInAS false, MemoryReserve 100
   VAR
      OpenFbChannel : Array[1..89] of Int;
      ClosedFbChannel : Array[1..89] of Int;
      HealthyChannel : Array[1..89] of Int;
      LocalModeChannel : Array[1..89] of Int;
      OpenCmdChannel : Array[1..89] of Int;
      CloseCmdChannel : Array[1..89] of Int;
   END_VAR
   VAR RETAIN
      TravelTimeout : Array[1..89] of Time;
      SeatBreakGrace : Array[1..89] of Time;
   END_VAR
BEGIN
   OpenFbChannel[1] := 1;
   OpenFbChannel[2] := 5;
   OpenFbChannel[3] := 9;
   OpenFbChannel[4] := 13;
   OpenFbChannel[5] := 17;
   OpenFbChannel[6] := 21;
   OpenFbChannel[7] := 25;
   OpenFbChannel[8] := 29;
   OpenFbChannel[9] := 33;
   OpenFbChannel[10] := 37;
   OpenFbChannel[11] := 41;
   OpenFbChannel[12] := 45;
   OpenFbChannel[13] := 49;
   OpenFbChannel[14] := 53;
   OpenFbChannel[15] := 57;
   OpenFbChannel[16] := 61;
   OpenFbChannel[17] := 65;
   OpenFbChannel[18] := 69;
   OpenFbChannel[19] := 73;
   OpenFbChannel[20] := 77;
   OpenFbChannel[21] := 81;
   OpenFbChannel[22] := 85;
   OpenFbChannel[23] := 89;
   OpenFbChannel[24] := 93;
   OpenFbChannel[25] := 97;
   OpenFbChannel[26] := 101;
   OpenFbChannel[27] := 105;
   OpenFbChannel[28] := 113;
   OpenFbChannel[29] := 117;
   OpenFbChannel[30] := 121;
   OpenFbChannel[31] := 125;
   OpenFbChannel[32] := 129;
   OpenFbChannel[33] := 133;
   OpenFbChannel[34] := 137;
   OpenFbChannel[35] := 141;
   OpenFbChannel[36] := 145;
   OpenFbChannel[37] := 149;
   OpenFbChannel[38] := 153;
   OpenFbChannel[39] := 157;
   OpenFbChannel[40] := 161;
   OpenFbChannel[41] := 165;
   OpenFbChannel[42] := 169;
   OpenFbChannel[43] := 173;
   OpenFbChannel[44] := 177;
   OpenFbChannel[45] := 181;
   OpenFbChannel[46] := 185;
   OpenFbChannel[47] := 189;
   OpenFbChannel[48] := 193;
   OpenFbChannel[49] := 197;
   OpenFbChannel[50] := 201;
   OpenFbChannel[51] := 205;
   OpenFbChannel[52] := 209;
   OpenFbChannel[53] := 213;
   OpenFbChannel[54] := 217;
   OpenFbChannel[55] := 225;
   OpenFbChannel[56] := 229;
   OpenFbChannel[57] := 233;
   OpenFbChannel[58] := 237;
   OpenFbChannel[59] := 241;
   OpenFbChannel[60] := 245;
   OpenFbChannel[61] := 249;
   OpenFbChannel[62] := 253;
   OpenFbChannel[63] := 257;
   OpenFbChannel[64] := 261;
   OpenFbChannel[65] := 265;
   OpenFbChannel[66] := 269;
   OpenFbChannel[67] := 273;
   OpenFbChannel[68] := 277;
   OpenFbChannel[69] := 281;
   OpenFbChannel[70] := 285;
   OpenFbChannel[71] := 289;
   OpenFbChannel[72] := 293;
   OpenFbChannel[73] := 297;
   OpenFbChannel[74] := 301;
   OpenFbChannel[75] := 305;
   OpenFbChannel[76] := 309;
   OpenFbChannel[77] := 313;
   OpenFbChannel[78] := 317;
   OpenFbChannel[79] := 321;
   OpenFbChannel[80] := 325;
   OpenFbChannel[81] := 329;
   OpenFbChannel[82] := 333;
   OpenFbChannel[83] := 337;
   OpenFbChannel[84] := 341;
   OpenFbChannel[85] := 345;
   OpenFbChannel[86] := 349;
   OpenFbChannel[87] := 353;
   OpenFbChannel[88] := 357;
   OpenFbChannel[89] := 361;
   ClosedFbChannel[1] := 2;
   ClosedFbChannel[2] := 6;
   ClosedFbChannel[3] := 10;
   ClosedFbChannel[4] := 14;
   ClosedFbChannel[5] := 18;
   ClosedFbChannel[6] := 22;
   ClosedFbChannel[7] := 26;
   ClosedFbChannel[8] := 30;
   ClosedFbChannel[9] := 34;
   ClosedFbChannel[10] := 38;
   ClosedFbChannel[11] := 42;
   ClosedFbChannel[12] := 46;
   ClosedFbChannel[13] := 50;
   ClosedFbChannel[14] := 54;
   ClosedFbChannel[15] := 58;
   ClosedFbChannel[16] := 62;
   ClosedFbChannel[17] := 66;
   ClosedFbChannel[18] := 70;
   ClosedFbChannel[19] := 74;
   ClosedFbChannel[20] := 78;
   ClosedFbChannel[21] := 82;
   ClosedFbChannel[22] := 86;
   ClosedFbChannel[23] := 90;
   ClosedFbChannel[24] := 94;
   ClosedFbChannel[25] := 98;
   ClosedFbChannel[26] := 102;
   ClosedFbChannel[27] := 106;
   ClosedFbChannel[28] := 114;
   ClosedFbChannel[29] := 118;
   ClosedFbChannel[30] := 122;
   ClosedFbChannel[31] := 126;
   ClosedFbChannel[32] := 130;
   ClosedFbChannel[33] := 134;
   ClosedFbChannel[34] := 138;
   ClosedFbChannel[35] := 142;
   ClosedFbChannel[36] := 146;
   ClosedFbChannel[37] := 150;
   ClosedFbChannel[38] := 154;
   ClosedFbChannel[39] := 158;
   ClosedFbChannel[40] := 162;
   ClosedFbChannel[41] := 166;
   ClosedFbChannel[42] := 170;
   ClosedFbChannel[43] := 174;
   ClosedFbChannel[44] := 178;
   ClosedFbChannel[45] := 182;
   ClosedFbChannel[46] := 186;
   ClosedFbChannel[47] := 190;
   ClosedFbChannel[48] := 194;
   ClosedFbChannel[49] := 198;
   ClosedFbChannel[50] := 202;
   ClosedFbChannel[51] := 206;
   ClosedFbChannel[52] := 210;
   ClosedFbChannel[53] := 214;
   ClosedFbChannel[54] := 218;
   ClosedFbChannel[55] := 226;
   ClosedFbChannel[56] := 230;
   ClosedFbChannel[57] := 234;
   ClosedFbChannel[58] := 238;
   ClosedFbChannel[59] := 242;
   ClosedFbChannel[60] := 246;
   ClosedFbChannel[61] := 250;
   ClosedFbChannel[62] := 254;
   ClosedFbChannel[63] := 258;
   ClosedFbChannel[64] := 262;
   ClosedFbChannel[65] := 266;
   ClosedFbChannel[66] := 270;
   ClosedFbChannel[67] := 274;
   ClosedFbChannel[68] := 278;
   ClosedFbChannel[69] := 282;
   ClosedFbChannel[70] := 286;
   ClosedFbChannel[71] := 290;
   ClosedFbChannel[72] := 294;
   ClosedFbChannel[73] := 298;
   ClosedFbChannel[74] := 302;
   ClosedFbChannel[75] := 306;
   ClosedFbChannel[76] := 310;
   ClosedFbChannel[77] := 314;
   ClosedFbChannel[78] := 318;
   ClosedFbChannel[79] := 322;
   ClosedFbChannel[80] := 326;
   ClosedFbChannel[81] := 330;
   ClosedFbChannel[82] := 334;
   ClosedFbChannel[83] := 338;
   ClosedFbChannel[84] := 342;
   ClosedFbChannel[85] := 346;
   ClosedFbChannel[86] := 350;
   ClosedFbChannel[87] := 354;
   ClosedFbChannel[88] := 358;
   ClosedFbChannel[89] := 362;
   HealthyChannel[1] := 3;
   HealthyChannel[2] := 7;
   HealthyChannel[3] := 11;
   HealthyChannel[4] := 15;
   HealthyChannel[5] := 19;
   HealthyChannel[6] := 23;
   HealthyChannel[7] := 27;
   HealthyChannel[8] := 31;
   HealthyChannel[9] := 35;
   HealthyChannel[10] := 39;
   HealthyChannel[11] := 43;
   HealthyChannel[12] := 47;
   HealthyChannel[13] := 51;
   HealthyChannel[14] := 55;
   HealthyChannel[15] := 59;
   HealthyChannel[16] := 63;
   HealthyChannel[17] := 67;
   HealthyChannel[18] := 71;
   HealthyChannel[19] := 75;
   HealthyChannel[20] := 79;
   HealthyChannel[21] := 83;
   HealthyChannel[22] := 87;
   HealthyChannel[23] := 91;
   HealthyChannel[24] := 95;
   HealthyChannel[25] := 99;
   HealthyChannel[26] := 103;
   HealthyChannel[27] := 107;
   HealthyChannel[28] := 115;
   HealthyChannel[29] := 119;
   HealthyChannel[30] := 123;
   HealthyChannel[31] := 127;
   HealthyChannel[32] := 131;
   HealthyChannel[33] := 135;
   HealthyChannel[34] := 139;
   HealthyChannel[35] := 143;
   HealthyChannel[36] := 147;
   HealthyChannel[37] := 151;
   HealthyChannel[38] := 155;
   HealthyChannel[39] := 159;
   HealthyChannel[40] := 163;
   HealthyChannel[41] := 167;
   HealthyChannel[42] := 171;
   HealthyChannel[43] := 175;
   HealthyChannel[44] := 179;
   HealthyChannel[45] := 183;
   HealthyChannel[46] := 187;
   HealthyChannel[47] := 191;
   HealthyChannel[48] := 195;
   HealthyChannel[49] := 199;
   HealthyChannel[50] := 203;
   HealthyChannel[51] := 207;
   HealthyChannel[52] := 211;
   HealthyChannel[53] := 215;
   HealthyChannel[54] := 219;
   HealthyChannel[55] := 227;
   HealthyChannel[56] := 231;
   HealthyChannel[57] := 235;
   HealthyChannel[58] := 239;
   HealthyChannel[59] := 243;
   HealthyChannel[60] := 247;
   HealthyChannel[61] := 251;
   HealthyChannel[62] := 255;
   HealthyChannel[63] := 259;
   HealthyChannel[64] := 263;
   HealthyChannel[65] := 267;
   HealthyChannel[66] := 271;
   HealthyChannel[67] := 275;
   HealthyChannel[68] := 279;
   HealthyChannel[69] := 283;
   HealthyChannel[70] := 287;
   HealthyChannel[71] := 291;
   HealthyChannel[72] := 295;
   HealthyChannel[73] := 299;
   HealthyChannel[74] := 303;
   HealthyChannel[75] := 307;
   HealthyChannel[76] := 311;
   HealthyChannel[77] := 315;
   HealthyChannel[78] := 319;
   HealthyChannel[79] := 323;
   HealthyChannel[80] := 327;
   HealthyChannel[81] := 331;
   HealthyChannel[82] := 335;
   HealthyChannel[83] := 339;
   HealthyChannel[84] := 343;
   HealthyChannel[85] := 347;
   HealthyChannel[86] := 351;
   HealthyChannel[87] := 355;
   HealthyChannel[88] := 359;
   HealthyChannel[89] := 363;
   LocalModeChannel[1] := 4;
   LocalModeChannel[2] := 8;
   LocalModeChannel[3] := 12;
   LocalModeChannel[4] := 16;
   LocalModeChannel[5] := 20;
   LocalModeChannel[6] := 24;
   LocalModeChannel[7] := 28;
   LocalModeChannel[8] := 32;
   LocalModeChannel[9] := 36;
   LocalModeChannel[10] := 40;
   LocalModeChannel[11] := 44;
   LocalModeChannel[12] := 48;
   LocalModeChannel[13] := 52;
   LocalModeChannel[14] := 56;
   LocalModeChannel[15] := 60;
   LocalModeChannel[16] := 64;
   LocalModeChannel[17] := 68;
   LocalModeChannel[18] := 72;
   LocalModeChannel[19] := 76;
   LocalModeChannel[20] := 80;
   LocalModeChannel[21] := 84;
   LocalModeChannel[22] := 88;
   LocalModeChannel[23] := 92;
   LocalModeChannel[24] := 96;
   LocalModeChannel[25] := 100;
   LocalModeChannel[26] := 104;
   LocalModeChannel[27] := 108;
   LocalModeChannel[28] := 116;
   LocalModeChannel[29] := 120;
   LocalModeChannel[30] := 124;
   LocalModeChannel[31] := 128;
   LocalModeChannel[32] := 132;
   LocalModeChannel[33] := 136;
   LocalModeChannel[34] := 140;
   LocalModeChannel[35] := 144;
   LocalModeChannel[36] := 148;
   LocalModeChannel[37] := 152;
   LocalModeChannel[38] := 156;
   LocalModeChannel[39] := 160;
   LocalModeChannel[40] := 164;
   LocalModeChannel[41] := 168;
   LocalModeChannel[42] := 172;
   LocalModeChannel[43] := 176;
   LocalModeChannel[44] := 180;
   LocalModeChannel[45] := 184;
   LocalModeChannel[46] := 188;
   LocalModeChannel[47] := 192;
   LocalModeChannel[48] := 196;
   LocalModeChannel[49] := 200;
   LocalModeChannel[50] := 204;
   LocalModeChannel[51] := 208;
   LocalModeChannel[52] := 212;
   LocalModeChannel[53] := 216;
   LocalModeChannel[54] := 220;
   LocalModeChannel[55] := 228;
   LocalModeChannel[56] := 232;
   LocalModeChannel[57] := 236;
   LocalModeChannel[58] := 240;
   LocalModeChannel[59] := 244;
   LocalModeChannel[60] := 248;
   LocalModeChannel[61] := 252;
   LocalModeChannel[62] := 256;
   LocalModeChannel[63] := 260;
   LocalModeChannel[64] := 264;
   LocalModeChannel[65] := 268;
   LocalModeChannel[66] := 272;
   LocalModeChannel[67] := 276;
   LocalModeChannel[68] := 280;
   LocalModeChannel[69] := 284;
   LocalModeChannel[70] := 288;
   LocalModeChannel[71] := 292;
   LocalModeChannel[72] := 296;
   LocalModeChannel[73] := 300;
   LocalModeChannel[74] := 304;
   LocalModeChannel[75] := 308;
   LocalModeChannel[76] := 312;
   LocalModeChannel[77] := 316;
   LocalModeChannel[78] := 320;
   LocalModeChannel[79] := 324;
   LocalModeChannel[80] := 328;
   LocalModeChannel[81] := 332;
   LocalModeChannel[82] := 336;
   LocalModeChannel[83] := 340;
   LocalModeChannel[84] := 344;
   LocalModeChannel[85] := 348;
   LocalModeChannel[86] := 352;
   LocalModeChannel[87] := 356;
   LocalModeChannel[88] := 360;
   LocalModeChannel[89] := 364;
   OpenCmdChannel[1] := 1;
   OpenCmdChannel[2] := 3;
   OpenCmdChannel[3] := 5;
   OpenCmdChannel[4] := 7;
   OpenCmdChannel[5] := 9;
   OpenCmdChannel[6] := 11;
   OpenCmdChannel[7] := 13;
   OpenCmdChannel[8] := 15;
   OpenCmdChannel[9] := 17;
   OpenCmdChannel[10] := 19;
   OpenCmdChannel[11] := 21;
   OpenCmdChannel[12] := 23;
   OpenCmdChannel[13] := 25;
   OpenCmdChannel[14] := 27;
   OpenCmdChannel[15] := 29;
   OpenCmdChannel[16] := 31;
   OpenCmdChannel[17] := 33;
   OpenCmdChannel[18] := 35;
   OpenCmdChannel[19] := 37;
   OpenCmdChannel[20] := 39;
   OpenCmdChannel[21] := 41;
   OpenCmdChannel[22] := 43;
   OpenCmdChannel[23] := 45;
   OpenCmdChannel[24] := 47;
   OpenCmdChannel[25] := 49;
   OpenCmdChannel[26] := 51;
   OpenCmdChannel[27] := 53;
   OpenCmdChannel[28] := 65;
   OpenCmdChannel[29] := 67;
   OpenCmdChannel[30] := 69;
   OpenCmdChannel[31] := 71;
   OpenCmdChannel[32] := 73;
   OpenCmdChannel[33] := 75;
   OpenCmdChannel[34] := 77;
   OpenCmdChannel[35] := 79;
   OpenCmdChannel[36] := 81;
   OpenCmdChannel[37] := 83;
   OpenCmdChannel[38] := 85;
   OpenCmdChannel[39] := 87;
   OpenCmdChannel[40] := 89;
   OpenCmdChannel[41] := 91;
   OpenCmdChannel[42] := 93;
   OpenCmdChannel[43] := 95;
   OpenCmdChannel[44] := 97;
   OpenCmdChannel[45] := 99;
   OpenCmdChannel[46] := 101;
   OpenCmdChannel[47] := 103;
   OpenCmdChannel[48] := 105;
   OpenCmdChannel[49] := 107;
   OpenCmdChannel[50] := 109;
   OpenCmdChannel[51] := 111;
   OpenCmdChannel[52] := 113;
   OpenCmdChannel[53] := 115;
   OpenCmdChannel[54] := 117;
   OpenCmdChannel[55] := 129;
   OpenCmdChannel[56] := 131;
   OpenCmdChannel[57] := 133;
   OpenCmdChannel[58] := 135;
   OpenCmdChannel[59] := 137;
   OpenCmdChannel[60] := 139;
   OpenCmdChannel[61] := 141;
   OpenCmdChannel[62] := 143;
   OpenCmdChannel[63] := 145;
   OpenCmdChannel[64] := 147;
   OpenCmdChannel[65] := 149;
   OpenCmdChannel[66] := 151;
   OpenCmdChannel[67] := 153;
   OpenCmdChannel[68] := 155;
   OpenCmdChannel[69] := 157;
   OpenCmdChannel[70] := 159;
   OpenCmdChannel[71] := 161;
   OpenCmdChannel[72] := 163;
   OpenCmdChannel[73] := 165;
   OpenCmdChannel[74] := 167;
   OpenCmdChannel[75] := 169;
   OpenCmdChannel[76] := 171;
   OpenCmdChannel[77] := 173;
   OpenCmdChannel[78] := 175;
   OpenCmdChannel[79] := 177;
   OpenCmdChannel[80] := 179;
   OpenCmdChannel[81] := 181;
   OpenCmdChannel[82] := 183;
   OpenCmdChannel[83] := 185;
   OpenCmdChannel[84] := 187;
   OpenCmdChannel[85] := 189;
   OpenCmdChannel[86] := 191;
   OpenCmdChannel[87] := 193;
   OpenCmdChannel[88] := 195;
   OpenCmdChannel[89] := 197;
   CloseCmdChannel[1] := 2;
   CloseCmdChannel[2] := 4;
   CloseCmdChannel[3] := 6;
   CloseCmdChannel[4] := 8;
   CloseCmdChannel[5] := 10;
   CloseCmdChannel[6] := 12;
   CloseCmdChannel[7] := 14;
   CloseCmdChannel[8] := 16;
   CloseCmdChannel[9] := 18;
   CloseCmdChannel[10] := 20;
   CloseCmdChannel[11] := 22;
   CloseCmdChannel[12] := 24;
   CloseCmdChannel[13] := 26;
   CloseCmdChannel[14] := 28;
   CloseCmdChannel[15] := 30;
   CloseCmdChannel[16] := 32;
   CloseCmdChannel[17] := 34;
   CloseCmdChannel[18] := 36;
   CloseCmdChannel[19] := 38;
   CloseCmdChannel[20] := 40;
   CloseCmdChannel[21] := 42;
   CloseCmdChannel[22] := 44;
   CloseCmdChannel[23] := 46;
   CloseCmdChannel[24] := 48;
   CloseCmdChannel[25] := 50;
   CloseCmdChannel[26] := 52;
   CloseCmdChannel[27] := 54;
   CloseCmdChannel[28] := 66;
   CloseCmdChannel[29] := 68;
   CloseCmdChannel[30] := 70;
   CloseCmdChannel[31] := 72;
   CloseCmdChannel[32] := 74;
   CloseCmdChannel[33] := 76;
   CloseCmdChannel[34] := 78;
   CloseCmdChannel[35] := 80;
   CloseCmdChannel[36] := 82;
   CloseCmdChannel[37] := 84;
   CloseCmdChannel[38] := 86;
   CloseCmdChannel[39] := 88;
   CloseCmdChannel[40] := 90;
   CloseCmdChannel[41] := 92;
   CloseCmdChannel[42] := 94;
   CloseCmdChannel[43] := 96;
   CloseCmdChannel[44] := 98;
   CloseCmdChannel[45] := 100;
   CloseCmdChannel[46] := 102;
   CloseCmdChannel[47] := 104;
   CloseCmdChannel[48] := 106;
   CloseCmdChannel[49] := 108;
   CloseCmdChannel[50] := 110;
   CloseCmdChannel[51] := 112;
   CloseCmdChannel[52] := 114;
   CloseCmdChannel[53] := 116;
   CloseCmdChannel[54] := 118;
   CloseCmdChannel[55] := 130;
   CloseCmdChannel[56] := 132;
   CloseCmdChannel[57] := 134;
   CloseCmdChannel[58] := 136;
   CloseCmdChannel[59] := 138;
   CloseCmdChannel[60] := 140;
   CloseCmdChannel[61] := 142;
   CloseCmdChannel[62] := 144;
   CloseCmdChannel[63] := 146;
   CloseCmdChannel[64] := 148;
   CloseCmdChannel[65] := 150;
   CloseCmdChannel[66] := 152;
   CloseCmdChannel[67] := 154;
   CloseCmdChannel[68] := 156;
   CloseCmdChannel[69] := 158;
   CloseCmdChannel[70] := 160;
   CloseCmdChannel[71] := 162;
   CloseCmdChannel[72] := 164;
   CloseCmdChannel[73] := 166;
   CloseCmdChannel[74] := 168;
   CloseCmdChannel[75] := 170;
   CloseCmdChannel[76] := 172;
   CloseCmdChannel[77] := 174;
   CloseCmdChannel[78] := 176;
   CloseCmdChannel[79] := 178;
   CloseCmdChannel[80] := 180;
   CloseCmdChannel[81] := 182;
   CloseCmdChannel[82] := 184;
   CloseCmdChannel[83] := 186;
   CloseCmdChannel[84] := 188;
   CloseCmdChannel[85] := 190;
   CloseCmdChannel[86] := 192;
   CloseCmdChannel[87] := 194;
   CloseCmdChannel[88] := 196;
   CloseCmdChannel[89] := 198;
   TravelTimeout[1..89] := T#60s;
   SeatBreakGrace[1..89] := T#10s;
END_DATA_BLOCK

DATA_BLOCK "Valve_Meta_DB"   // DB11
{ S7_Optimized_Access := 'TRUE' }
VERSION : 0.1
// stored: AutoNumber true, IsOnlyStoredInLoadMemory false, IsRetainMemResEnabled false, IsWriteProtectedInAS false, MemoryReserve 100
   VAR
      "Name" : Array[1..89] of String[20];
      Location : Array[1..89] of String[20];
      CmNo : Array[1..89] of String[6];
      VTag : Array[1..89] of String[12];
      SysName : Array[1..89] of String[12];
      FuncName : Array[1..89] of String[22];
      AftTblName : Array[1..14] of String[20];
      ErTblName : Array[1..14] of String[20];
      FwdTblName : Array[1..14] of String[20];
      AftTblLoc : Array[1..14] of String[20];
      ErTblLoc : Array[1..14] of String[20];
      FwdTblLoc : Array[1..14] of String[20];
      AftTblCmNo : Array[1..14] of String[6];
      ErTblCmNo : Array[1..14] of String[6];
      FwdTblCmNo : Array[1..14] of String[6];
      AftTblVTag : Array[1..14] of String[12];
      ErTblVTag : Array[1..14] of String[12];
      FwdTblVTag : Array[1..14] of String[12];
      AftTblFunc : Array[1..14] of String[22];
      ErTblFunc : Array[1..14] of String[22];
      FwdTblFunc : Array[1..14] of String[22];
      CfgTblName : Array[1..16] of String[20];
      CfgTblLoc : Array[1..16] of String[20];
      CfgTblCmNo : Array[1..16] of String[6];
      CfgTblVTag : Array[1..16] of String[12];
      CfgTblSys : Array[1..16] of String[12];
      CfgTblFunc : Array[1..16] of String[22];
      SelCmNo : String[6];
      SelVTag : String[12];
   END_VAR
BEGIN
   Location[1..2] := 'DB tank';
   Location[3] := 'Main line';
   Location[4] := 'Aft peak C';
   Location[5] := 'Aft peak';
   Location[6] := 'Aft peak P';
   Location[7] := 'Aft peak S';
   Location[8..13] := 'DB tank';
   Location[14..15] := 'Cross line';
   Location[16..17] := 'Pump 2';
   Location[18] := 'Main line';
   Location[19] := 'Pump 2';
   Location[20] := 'Pump 1';
   Location[21] := 'Bilge tie';
   Location[22] := 'Bilge system tie';
   Location[23..24] := 'Pump 2 discharge';
   Location[25] := 'Tank branch';
   Location[26] := 'Main line';
   Location[27] := 'Cross line';
   Location[28] := 'Bow thruster room';
   Location[29..30] := 'Hold 4';
   Location[31..32] := 'Hold 3';
   Location[33] := 'ER';
   Location[34] := 'ER/Pipe void';
   Location[35] := 'Pipe void aft';
   Location[36..37] := 'Engine Room';
   Location[38..39] := 'Hold 2';
   Location[40..41] := 'Hold 1';
   Location[42] := 'ER';
   Location[43] := 'Pump suction';
   Location[44] := 'ER';
   Location[45] := 'Void Deck';
   Location[46] := 'Pipe void aft';
   Location[47..48] := 'Hold 5';
   Location[49..50] := 'Discharge';
   Location[51] := 'Fire main';
   Location[52] := 'Fire line';
   Location[53] := 'Bilge Fire Pump 2';
   Location[54] := 'Bilge Fire Pump 1';
   Location[55] := 'TK6 High P';
   Location[56..57] := 'Manifold';
   Location[58] := 'TK5 Wing P';
   Location[59] := 'TK4 DB';
   Location[60] := 'Manifold';
   Location[61] := 'TK5 DB P';
   Location[62] := 'Manifold';
   Location[63] := 'TK3 Wing S';
   Location[64..66] := 'Manifold';
   Location[67] := 'TK2 Wing P';
   Location[68] := 'TK1 DB C';
   Location[69] := 'Main line';
   Location[70] := 'TK2 High C';
   Location[71] := 'Main line';
   Location[72] := 'TK2 Wing S';
   Location[73] := 'Fwd peak';
   Location[74] := 'Main line';
   Location[75] := 'Fwd peak';
   Location[76] := 'TK3 Wing P';
   Location[77..78] := 'Manifold';
   Location[79] := 'TK4 Wing P';
   Location[80] := 'TK4 Wing S';
   Location[81..82] := 'Manifold';
   Location[83] := 'TK3 DB';
   Location[84] := 'Cross line';
   Location[85..87] := 'Cross-over manifold';
   Location[89] := 'Cross-over manifold';
   CmNo[1] := 'CM25';
   CmNo[2] := 'CM26';
   CmNo[3] := 'CM50';
   CmNo[4] := 'CM51';
   CmNo[5] := 'CM52';
   CmNo[6] := 'CM53';
   CmNo[7] := 'CM54';
   CmNo[8] := 'CM55';
   CmNo[9] := 'CM56';
   CmNo[10] := 'CM57';
   CmNo[11] := 'CM58';
   CmNo[12] := 'CM59';
   CmNo[13] := 'CM60';
   CmNo[14] := 'CM67';
   CmNo[15] := 'CM68';
   CmNo[16] := 'CM69';
   CmNo[17] := 'CM70';
   CmNo[18] := 'CM71';
   CmNo[19] := 'CM72';
   CmNo[20] := 'CM78';
   CmNo[21] := 'CM79';
   CmNo[22] := 'CM80';
   CmNo[23] := 'CM81';
   CmNo[24] := 'CM82';
   CmNo[25] := 'CM83';
   CmNo[26] := 'CM84';
   CmNo[27] := 'CM85';
   CmNo[28] := 'CM01';
   CmNo[29] := 'CM02';
   CmNo[30] := 'CM03';
   CmNo[31] := 'CM04';
   CmNo[32] := 'CM05';
   CmNo[33] := 'CM06';
   CmNo[34] := 'CM07';
   CmNo[35] := 'CM08';
   CmNo[36] := 'CM09';
   CmNo[37] := 'CM10';
   CmNo[38] := 'CM11';
   CmNo[39] := 'CM12';
   CmNo[40] := 'CM13';
   CmNo[41] := 'CM14';
   CmNo[42] := 'CM15';
   CmNo[43] := 'CM16';
   CmNo[44] := 'CM17';
   CmNo[45] := 'CM18';
   CmNo[46] := 'CM19';
   CmNo[47] := 'CM20';
   CmNo[48] := 'CM21';
   CmNo[49] := 'CM23';
   CmNo[50] := 'CM24';
   CmNo[51] := 'CM94';
   CmNo[52] := 'CM95';
   CmNo[53] := 'CM96';
   CmNo[54] := 'CM97';
   CmNo[55] := 'CM27';
   CmNo[56] := 'CM28';
   CmNo[57] := 'CM29';
   CmNo[58] := 'CM30';
   CmNo[59] := 'CM31';
   CmNo[60] := 'CM32';
   CmNo[61] := 'CM33';
   CmNo[62] := 'CM34';
   CmNo[63] := 'CM35';
   CmNo[64] := 'CM36';
   CmNo[65] := 'CM37';
   CmNo[66] := 'CM38';
   CmNo[67] := 'CM39';
   CmNo[68] := 'CM40';
   CmNo[69] := 'CM41';
   CmNo[70] := 'CM42';
   CmNo[71] := 'CM43';
   CmNo[72] := 'CM44';
   CmNo[73] := 'CM45';
   CmNo[74] := 'CM46';
   CmNo[75] := 'CM47';
   CmNo[76] := 'CM48';
   CmNo[77] := 'CM49';
   CmNo[78] := 'CM61';
   CmNo[79] := 'CM62';
   CmNo[80] := 'CM63';
   CmNo[81] := 'CM64';
   CmNo[82] := 'CM65';
   CmNo[83] := 'CM66';
   CmNo[84] := 'CM77';
   CmNo[85] := 'CM86';
   CmNo[86] := 'CM87';
   CmNo[87] := 'CM88';
   CmNo[88] := 'CM89';
   CmNo[89] := 'CM90';
   VTag[1] := '11-020-A1';
   VTag[2] := '11-021-A1';
   VTag[3] := '11-008-A1';
   VTag[4] := '11-009-A1';
   VTag[5] := '11-010-A1';
   VTag[6] := '11-060-A1';
   VTag[7] := '11-061-A1';
   VTag[8] := '11-024-A2';
   VTag[9] := '11-025-A2';
   VTag[10] := '11-028-A1';
   VTag[11] := '11-029-A1';
   VTag[12] := '11-022-A2';
   VTag[13] := '11-023-A2';
   VTag[14] := '11-001-A2';
   VTag[15] := '11-004-A1';
   VTag[16] := '11-002-A2';
   VTag[17] := '11-002-A4';
   VTag[18] := '11-005-A1';
   VTag[19] := '11-006-A1';
   VTag[20] := '11-011-A1';
   VTag[21] := '11-011-A3';
   VTag[22] := '11-011-A4';
   VTag[23] := '11-012-A1';
   VTag[24] := '11-012-A3';
   VTag[25] := '11-015-A1';
   VTag[26] := '11-016-A1';
   VTag[27] := '11-003-A1';
   VTag[28] := '10-041-A1';
   VTag[29] := '10-017-A1';
   VTag[30] := '10-018-A1';
   VTag[31] := '10-021-A1';
   VTag[32] := '10-022-A1';
   VTag[33] := '10-007-A1';
   VTag[34] := '10-009-A1';
   VTag[35] := '10-012-A1';
   VTag[36] := '10-001-A1';
   VTag[37] := '10-002-A1';
   VTag[38] := '10-025-A1';
   VTag[39] := '10-026-A1';
   VTag[40] := '10-034-A1';
   VTag[41] := '10-035-A1';
   VTag[42] := '10-003-A1';
   VTag[43] := '10-004-A1';
   VTag[44] := '10-005-A1';
   VTag[45] := '10-001-A2';
   VTag[46] := '10-013-A1';
   VTag[47] := '10-010-A1';
   VTag[48] := '10-011-A1';
   VTag[49] := '10-046-A1';
   VTag[50] := '10-047-A2';
   VTag[51] := '20-023-A1';
   VTag[52] := '20-025-A1';
   VTag[53] := '20-022-A1';
   VTag[54] := '20-024-A1';
   VTag[55] := '11-030-A1';
   VTag[56] := '11-031-A1';
   VTag[57] := '11-032-A1';
   VTag[58] := '11-033-A1';
   VTag[59] := '11-034-A2';
   VTag[60] := '11-035-A1';
   VTag[61] := '11-036-A1';
   VTag[62] := '11-037-A1';
   VTag[63] := '11-046-A1';
   VTag[64] := '11-047-A2';
   VTag[65] := '11-048-A1';
   VTag[66] := '11-049-A1';
   VTag[67] := '11-050-A1';
   VTag[68] := '11-051-A1';
   VTag[69] := '11-052-A1';
   VTag[70] := '11-053-A1';
   VTag[71] := '11-054-A2';
   VTag[72] := '11-055-A1';
   VTag[73] := '11-056-A1';
   VTag[74] := '11-057-A1';
   VTag[75] := '11-058-A1';
   VTag[76] := '11-042-A1';
   VTag[77] := '11-043-A1';
   VTag[78] := '11-043-A2';
   VTag[79] := '11-041-A2';
   VTag[80] := '11-039-A1';
   VTag[81] := '11-040-A1';
   VTag[82] := '11-044-A2';
   VTag[83] := '11-045-A2';
   VTag[84] := '11-014-A1';
   VTag[85] := '11-063-A1';
   VTag[86] := '11-064-A1';
   VTag[87] := '11-065-A1';
   VTag[88] := '11-066-A1';
   VTag[89] := '11-067-A1';
   SysName[1..27] := 'Ballast Aft';
   SysName[28..54] := 'Bilge';
   SysName[55..89] := 'Ballast Fwd';
   FuncName[1] := 'Filling';
   FuncName[2] := 'Suction';
   FuncName[3..5] := 'Isolation';
   FuncName[6..7] := 'Tank suction';
   FuncName[8] := 'Filling';
   FuncName[9..10] := 'Suction';
   FuncName[11] := 'Filling';
   FuncName[12] := 'Suction';
   FuncName[13] := 'Filling';
   FuncName[14..17] := 'Isolation';
   FuncName[18] := 'Distribution';
   FuncName[19] := 'Suction';
   FuncName[20] := 'Discharge';
   FuncName[21] := 'Cross connect';
   FuncName[22..27] := 'Isolation';
   FuncName[28..32] := 'Bilge suction';
   FuncName[33] := 'Suction';
   FuncName[34..35] := 'Isolation';
   FuncName[36] := 'Suction';
   FuncName[37] := 'Main suction';
   FuncName[38..41] := 'Bilge suction';
   FuncName[42] := 'Suction';
   FuncName[43] := 'Isolation';
   FuncName[44] := 'Suction';
   FuncName[45] := 'Bilge suction';
   FuncName[46] := 'Isolation';
   FuncName[47..48] := 'Bilge suction';
   FuncName[49..51] := 'Isolation';
   FuncName[52] := 'Fire/Bilge crossover';
   FuncName[53..54] := 'Seawater priming';
   FuncName[55] := 'Filling';
   FuncName[56..57] := 'Suction';
   FuncName[58..59] := 'Filling';
   FuncName[60] := 'Suction';
   FuncName[61] := 'Filling';
   FuncName[62] := 'Suction';
   FuncName[63] := 'Filling';
   FuncName[64..66] := 'Suction';
   FuncName[67..68] := 'Filling';
   FuncName[69] := 'Isolation';
   FuncName[70] := 'Filling';
   FuncName[71] := 'Isolation';
   FuncName[72..73] := 'Filling';
   FuncName[74] := 'Isolation';
   FuncName[75..76] := 'Filling';
   FuncName[77..78] := 'Suction';
   FuncName[79..80] := 'Filling';
   FuncName[81..82] := 'Suction';
   FuncName[83] := 'Filling';
   FuncName[84..87] := 'Isolation';
   FuncName[89] := 'Isolation';
END_DATA_BLOCK

DATA_BLOCK "Valves_DB"   // DB5
{ S7_Optimized_Access := 'TRUE' }
VERSION : 0.1
// stored: AutoNumber true, IsOnlyStoredInLoadMemory false, IsRetainMemResEnabled false, IsWriteProtectedInAS false, MemoryReserve 100
   VAR
      Valve : Array[1..89] of "Valve_IO";
      TotalOpen : Int;
      TotalClosed : Int;
      TotalTransit : Int;
      TotalFault : Int;
      TotalLocal : Int;
      TotalConfigured : Int;
      ErOpen : Int;
      ErClosed : Int;
      ErTransit : Int;
      ErFault : Int;
      ErLocal : Int;
      ErConfigured : Int;
      FwdOpen : Int;
      FwdClosed : Int;
      FwdTransit : Int;
      FwdFault : Int;
      FwdLocal : Int;
      FwdConfigured : Int;
      AftOpen : Int;
      AftClosed : Int;
      AftTransit : Int;
      AftFault : Int;
      AftLocal : Int;
      AftConfigured : Int;
      StateCode : Array[1..89] of Int;
      Stuck : Array[1..89] of Bool;
      Initialized : Array[1..89] of Bool;
      TimeoutOpenAlarm : Array[1..89] of Bool;
      TimeoutCloseAlarm : Array[1..89] of Bool;
      UnexpMove : Array[1..89] of Bool;
      DirFault : Array[1..89] of Bool;
      PosCode : Array[1..89] of Int;
      FaultCode : Array[1..89] of Int;
      CmdPos : Array[1..89] of Int;
      PrevOpenFB : Array[1..89] of Bool;
      PrevClosedFB : Array[1..89] of Bool;
      PosLostTmr : Array[1..89] of TON_TIME;
      DirTmr : Array[1..89] of TON_TIME;
      HwHealthy : Array[1..9] of Bool;
      W_Unhealthy : Array[0..5] of Word;
      W_Conflict : Array[0..5] of Word;
      W_FailOpen : Array[0..5] of Word;
      W_FailClose : Array[0..5] of Word;
      W_LossPos : Array[0..5] of Word;
      W_UnexpMove : Array[0..5] of Word;
      W_Local : Array[0..5] of Word;
      W_DirFault : Array[0..5] of Word;
      HwWord : Word;
      AftPage : Int;
      ErPage : Int;
      FwdPage : Int;
      AftTblState : Array[1..14] of Int;
      ErTblState : Array[1..14] of Int;
      FwdTblState : Array[1..14] of Int;
      AftTblNo : Array[1..14] of Int;
      ErTblNo : Array[1..14] of Int;
      FwdTblNo : Array[1..14] of Int;
      AftTblStateTxt : Array[1..14] of String[14];
      ErTblStateTxt : Array[1..14] of String[14];
      FwdTblStateTxt : Array[1..14] of String[14];
      AftTblTag : Array[1..14] of String[8];
      ErTblTag : Array[1..14] of String[8];
      FwdTblTag : Array[1..14] of String[8];
      CfgPage : Int;
      CfgTblNo : Array[1..16] of Int;
      CfgTblTag : Array[1..16] of String[8];
      CfgTblZone : Array[1..16] of String[12];
      CfgTblConfigured : Array[1..16] of Bool;
      CfgTblState : Array[1..16] of Int;
      CfgTblStateTxt : Array[1..16] of String[14];
      Clock_1Hz : Bool;
      ClockCounter : Int;
      SelIdx : Int;
      SelState : Int;
      SelHealthy : Bool;
      SelLocalMode : Bool;
      SelConfigured : Bool;
      DispCode : Array[1..89] of Int;
      Clock_Flash : Bool;
      HwInitDone : Bool;
   END_VAR
   VAR RETAIN
      ConfiguredRet : Array[1..89] of Bool;
   END_VAR
   VAR
      Clk1Tmr : TON_TIME;
      FlashTmr : TON_TIME;
      WinTmr : TON_TIME;
      PrevAftPage : Int;
      PrevErPage : Int;
      PrevFwdPage : Int;
      PrevCfgPage : Int;
      SelDirFault : Bool;
      SelCmdPos : Int;
      SelPosCode : Int;
      SelFaultCode : Int;
   END_VAR
BEGIN
END_DATA_BLOCK

DATA_BLOCK "HMI_Interface_DB"   // DB7
{ S7_Optimized_Access := 'TRUE' }
VERSION : 0.1
// stored: AutoNumber true, IsOnlyStoredInLoadMemory false, IsRetainMemResEnabled false, IsWriteProtectedInAS false, MemoryReserve 100
   VAR
      SelectedValveIndex : Int;
      OpenCmd : Bool;
      CloseCmd : Bool;
      OpenFB : Bool;
      ClosedFB : Bool;
      Healthy : Bool;
      LocalMode : Bool;
   END_VAR
BEGIN
END_DATA_BLOCK

DATA_BLOCK "IO_Buffer_DB"   // DB
{ S7_Optimized_Access := 'TRUE' }
VERSION : 0.1
// Abstract channel table: DI[1..368] covers all 23 DI16 modules across AFT/MID/FWD (7+7+9), DQ[1..208] covers all 13 DQ16 modules (4+4+5) - matches the confirmed BOM module counts. Index N here is OUR OWN channel numbering, not a real %I/%Q address - FC_IoMapper is the only place real physical addresses get referenced, once the hardware address assignment question (see FC_IoMapper header comment) is resolved.
// stored: AutoNumber true, IsOnlyStoredInLoadMemory false, IsRetainMemResEnabled false, IsWriteProtectedInAS false, MemoryReserve 100
   VAR
      DI : Array[1..368] of Bool;
      DQ : Array[1..208] of Bool;
   END_VAR
BEGIN
END_DATA_BLOCK

ORGANIZATION_BLOCK "Main"   // OB1, LAD, ProgramCycle
TITLE = "Main Program Sweep (Cycle)"
{ S7_Optimized_Access := 'TRUE' }
VERSION : 0.1
// stored: AutoNumber true, IsIECCheckEnabled false, SetENOAutomatically false
   VAR_INPUT
      Initial_Call : Bool;   // Initial call of this OB
      Remanence : Bool;   // =True, if remanent data are available
   END_VAR
BEGIN

REGION Network 1
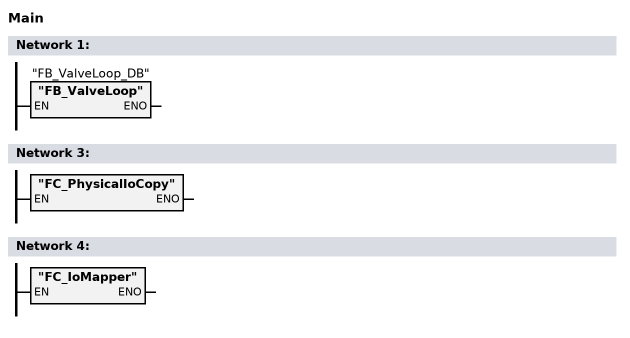
   RUNG wire#powerrail
      "FB_ValveLoop_DB"()
   END_RUNG
   // the same network as SCL:
   "FB_ValveLoop_DB"();   // "FB_ValveLoop"
END_REGION

REGION Network 3
   RUNG wire#powerrail
      "FC_PhysicalIoCopy"()
   END_RUNG
   // the same network as SCL:
   "FC_PhysicalIoCopy"();
END_REGION

REGION Network 4
   RUNG wire#powerrail
      "FC_IoMapper"()
   END_RUNG
   // the same network as SCL:
   "FC_IoMapper"();
END_REGION
END_ORGANIZATION_BLOCK

FUNCTION_BLOCK "FB_ValveLoop"   // FB4, SCL
{ S7_Optimized_Access := 'TRUE' }
VERSION : 0.1
// stored: AutoNumber true, IsIECCheckEnabled false, IsRetainMemResEnabled false, MemoryReserve 100, SetENOAutomatically false, UDAEnableTagReadback false
   VAR
      i { S7_SetPoint := 'True'} : Int;
      SimStep : Array[1..89] of Int;
   END_VAR
   VAR_TEMP
      tempOpen : Int;
      tempClosed : Int;
      tempTransit : Int;
      tempFault : Int;
      tempLocal : Int;
      tempConfigured : Int;
      tempErOpen : Int;
      tempErClosed : Int;
      tempErTransit : Int;
      tempErFault : Int;
      tempErLocal : Int;
      tempErConfigured : Int;
      tempFwdOpen : Int;
      tempFwdClosed : Int;
      tempFwdTransit : Int;
      tempFwdFault : Int;
      tempFwdLocal : Int;
      tempFwdConfigured : Int;
      tempAftOpen : Int;
      tempAftClosed : Int;
      tempAftTransit : Int;
      tempAftFault : Int;
      tempAftLocal : Int;
      tempAftConfigured : Int;
      j : Int;
      z : Int;
      idx : Int;
      base : Int;
      zStart : Int;
      zEnd : Int;
      tagStr : String[8];
      w : Int;
      "b" : Int;
      bitIdx : Int;
      packWord : Word;
      simStepAtStart : Int;
      sel : Int;
      travelPT : Time;
      seatPT : Time;
      winTick : Bool;
      doWindows : Bool;
   END_VAR
BEGIN

       #tempOpen := 0;
       #tempClosed := 0;
       #tempTransit := 0;
       #tempFault := 0;
       #tempLocal := 0;
       #tempConfigured := 0;
       #tempErOpen := 0;    #tempErClosed := 0;    #tempErTransit := 0;    #tempErFault := 0;    #tempErLocal := 0;    #tempErConfigured := 0;
       #tempFwdOpen := 0;   #tempFwdClosed := 0;   #tempFwdTransit := 0;   #tempFwdFault := 0;   #tempFwdLocal := 0;   #tempFwdConfigured := 0;
       #tempAftOpen := 0;   #tempAftClosed := 0;   #tempAftTransit := 0;   #tempAftFault := 0;   #tempAftLocal := 0;   #tempAftConfigured := 0;

               // Flash clocks — TIME based, not scan-count based.
       // The old version incremented a counter and toggled at >= 10, i.e. every TEN SCANS. That is
       // only 1 Hz if a scan takes 50 ms; the real scan is a few milliseconds, so it was toggling at
       // roughly 16 Hz and the popup's "1 Hz" fault flash was actually a fast flicker. A TON runs on
       // the CPU clock, so these are correct regardless of scan time.
       "Valves_DB".ClockCounter := 0;   // legacy scan counter, no longer used
       "Valves_DB".Clk1Tmr(IN := TRUE, PT := T#500MS);
       IF "Valves_DB".Clk1Tmr.Q THEN
           "Valves_DB".Clock_1Hz := NOT "Valves_DB".Clock_1Hz;   // a genuine 1 Hz now
           "Valves_DB".Clk1Tmr(IN := FALSE, PT := T#500MS);   // reset NOW, same scan
       END_IF;
       "Valves_DB".FlashTmr(IN := TRUE, PT := T#2S);
       IF "Valves_DB".FlashTmr.Q THEN
           "Valves_DB".Clock_Flash := NOT "Valves_DB".Clock_Flash;   // 0.25 Hz: 2 s on, 2 s off
           "Valves_DB".FlashTmr(IN := FALSE, PT := T#2S);   // reset NOW, same scan
       END_IF;
       // Self-referencing IN (IN := NOT Q) looked correct but never produced an observable
       // pulse: the moment the TON sets Q, the IN expression evaluates FALSE and the timer
       // clears Q again before the following IF can read it. Observed live 2026-08-19 -
       // Clock_Flash never went true (faulted valves showed steady position colour, no red
       // flash) and the table windows only ever refreshed when a page button was pressed.
       // Drive IN unconditionally TRUE and reset explicitly in the same scan instead.
       "Valves_DB".WinTmr(IN := TRUE, PT := T#200MS);
       #winTick := "Valves_DB".WinTmr.Q;   // latch before the reset clears it
       IF #winTick THEN
           "Valves_DB".WinTmr(IN := FALSE, PT := T#200MS);
       END_IF;

       // Hardware health starts healthy-until-told-otherwise, once per CPU start.
       //
       // This used to test "HwHealthy[1] AND [8] are both FALSE" as a stand-in for "nothing has been
       // set yet". That worked only while nothing drove those two bits - and they are bit 0 (PLC CPU
       // fault) and bit 7 (HMI heartbeat loss), both of which are due to be driven. The moment they
       // are, the sentinel becomes reachable in normal operation: one CPU fault alongside a lost
       // heartbeat would re-run this loop and reset all nine bits to healthy, silently taking the
       // three WORKING station alarms with it. Not a far-fetched pair either - a panel powered down
       // overnight holds heartbeat-lost on its own, so it needs only one CPU diagnostic beside it.
       //
       // HwInitDone says what is actually meant. It is NonRetain with no start value, so it is FALSE
       // on every CPU start and TRUE for the rest of that run - which is the real definition of
       // "first scan", and cannot be re-entered by live fault data no matter what drives the bits.
       // Keep it NonRetain even as other Valves_DB members become retentive: resetting on every
       // restart is the whole point of it.
       IF NOT "Valves_DB".HwInitDone THEN
           FOR #b := 1 TO 9 DO
               "Valves_DB".HwHealthy[#b] := TRUE;
           END_FOR;

           // Restore which valves were in service, from the retentive mirror. Without this the
           // whole plant came back UNCONFIGURED after any power cut: Configured is non-retentive
           // with no start value, so all 89 read FALSE, FC_IoMapper skipped every valve and
           // FB_ValveLoop refused every command - while the panel looked entirely normal. Nothing
           // on the ship answered until somebody knew to press CONFIGURE ALL.
           //
           // Restored here rather than anywhere else because this block is the only code that runs
           // exactly once per CPU start, before the 1..89 loop below saves the value straight back.
           // Order matters: restore first, then the loop's save is a no-op on this scan.
           FOR #b := 1 TO 89 DO
               "Valves_DB".Valve[#b].Configured := "Valves_DB".ConfiguredRet[#b];
           END_FOR;

           "Valves_DB".HwInitDone := TRUE;
       END_IF;

       // Remote I/O station health, from OB86 (RackOrStationFailure) via Diag_DB. HwHealthy[2..4]
       // are already wired to the System_Aft/Bilge/Fwd_RIO_Fault alarms through HwWord bits 1..3 -
       // those alarms have existed since the alarm set was generated and nothing has ever set them,
       // so a station could drop off PROFINET and the alarm built for exactly that stayed silent.
       //
       // Derived here every scan rather than written directly by OB86, because of the auto-init
       // immediately above: it fires whenever HwHealthy[1] and [8] are both FALSE, which is the
       // state at CPU startup. A station already down when the CPU starts would have OB86 set its
       // bit and then have that init wipe it in the same scan. Diag_DB is written by OB86 alone and
       // read here, so the ordering cannot lose a genuine station loss.
       //
       // Sense is inverted: HwHealthy TRUE means well, and HwWord sets its bit on NOT HwHealthy.
       "Valves_DB".HwHealthy[2] := NOT "Diag_DB".AftLost;
       "Valves_DB".HwHealthy[3] := NOT "Diag_DB".MidLost;
       "Valves_DB".HwHealthy[4] := NOT "Diag_DB".FwdLost;

       // I/O module diagnostics, from OB82 via Diag_DB - HwHealthy[5] is HwWord bit 4, which
       // already drives the System_IO_Module_Fault alarm. Added 2026-09-10 (item 37 bit 4).
       //
       // The acknowledge is consumed BEFORE HwHealthy[5] is computed, so a reset clears the alarm
       // in the same scan it is requested rather than leaving it up for one more. OB82 latches the
       // flag and never clears it - deliberately, because it cannot tell a fault appearing from one
       // going away without decoding IO_State, whose bit meanings are unconfirmed. See OB82.
       //
       // Consequence to expect on the panel: a module fault stays raised after the module recovers,
       // until someone acknowledges it. That is the safe direction and it is the intended behaviour,
       // not a bug to fix by making this self-clearing.
       IF "Diag_DB".ModuleFaultAck THEN
           "Diag_DB".ModuleFault := FALSE;
           "Diag_DB".ModuleFaultAck := FALSE;
       END_IF;
       "Valves_DB".HwHealthy[5] := NOT "Diag_DB".ModuleFault;

       FOR #i := 1 TO 89 DO
           // Keep the retentive mirror in step with the live flag, so whatever an engineer sets on
           // the Config screen survives the next blackout. One Bool copy per valve per scan.
           "Valves_DB".ConfiguredRet[#i] := "Valves_DB".Valve[#i].Configured;

           // Per-valve stroke times, replacing the compiled-in T#8S and T#5S. Both were simulation
           // numbers: real DN200-DN400 hydraulic valves stroke in 15-60s, and because the command is
           // MAINTAINED, an expiring timer drops the run latch and physically halts the valve rather
           // than merely raising an alarm. The 5s direction grace was the worse of the two, since it
           // arms the moment a valve is driven while still on its starting limit switch - which is
           // exactly what a large valve does for its first few seconds - so every normal stroke
           // raised a direction fault before the travel timeout ever got a chance.
           //
           // Zero guard is not paranoia: PT := T#0S expires on the very first scan, so a bad import
           // or a mis-typed panel entry would be worse than the 8 seconds this replaces. Falling back
           // to the generous default keeps a wrong number merely late rather than actively harmful.
           #travelPT := "Valve_Channels_DB".TravelTimeout[#i];
           IF #travelPT <= T#0S THEN #travelPT := T#60S; END_IF;
           #seatPT := "Valve_Channels_DB".SeatBreakGrace[#i];
           IF #seatPT <= T#0S THEN #seatPT := T#10S; END_IF;

           IF "Valves_DB".Valve[#i].Configured THEN
               // Snapshot BEFORE this scan's command/timer processing runs — needed by the
               // Unexpected Movement (F) guard below to tell a genuine idle-and-unexplained drop
               // apart from a normal command-triggered one (a fresh command sets SimStep 0->nonzero
               // in section 1; a completing travel sets it nonzero->0 in section 2 — comparing
               // only the post-scan value can't distinguish either from true idle-the-whole-scan).
               #simStepAtStart := #SimStep[#i];

               // Auto-initialize Healthy status to TRUE and Resting Position to CLOSED seat — but
               // ONLY the first scan a valve is ever seen, via the Initialized latch. Simulation-only
               // scaffolding (see the Initialized member's comment in Valves_DB): without this
               // one-time gate, this ran every scan and silently reset ClosedFB back to TRUE any time
               // a valve was idle with both feedbacks false — which is exactly the state Loss of
               // Position (E) needs to sustain for 2s to fire, so E could never actually trigger.
               //
               // Real-channel valves must NEVER have ClosedFB assumed here - only real hardware
               // feedback (via FC_IoMapper) may ever set it. Confirmed live via watch-table test
               // 2026-08-13: forcing a real valve's Configured=TRUE while its real DI already read
               // OpenFB=TRUE caused this block to also force ClosedFB=TRUE the same scan (assuming
               // "starts closed"), so both feedbacks were true at once and the double-indication
               // fault check below correctly tripped Healthy=FALSE for the wrong reason. Real valves
               // still get the one-time Healthy=TRUE start, just never the assumed position.
               IF NOT "Valves_DB".Initialized[#i] THEN
                   "Valves_DB".Initialized[#i] := TRUE;
                   // Real-channel valves get NOTHING seeded here. Healthy, OpenFB and ClosedFB are
                   // valve-owned signals - the valve reports them, the PLC only reads them - and
                   // FC_IoMapper fills all three from real hardware later in this very same scan.
                   // Seeding Healthy:=TRUE was harmless in effect (overwritten immediately) but it
                   // was still the PLC writing a signal it does not own. Removed 2026-08-15.
                   IF "Valve_Channels_DB".OpenFbChannel[#i] = 0
                      AND NOT "Valves_DB".Valve[#i].OpenFB AND NOT "Valves_DB".Valve[#i].ClosedFB
                      AND #SimStep[#i] = 0 THEN
                       "Valves_DB".Valve[#i].Healthy := TRUE;
                       "Valves_DB".Valve[#i].ClosedFB := TRUE;
                   END_IF;
               END_IF;

               // 1. Failsafe Command, real-channel latch, and Motion Simulation
               // A valve with a real DI channel assigned (Valve_Channels_DB.OpenFbChannel[i] > 0)
               // never gets its OpenFB/ClosedFB touched here or in Section 2 below - those come from
               // real hardware via FC_IoMapper instead. What THIS valve needs from a command is a
               // sustained "run" output (OpenValve/CloseValve) for FC_IoMapper to drive to the real
               // DQ, latched until the real limit switch confirms arrival (see the block right after
               // this one) or a timeout gives up (Section 2, real-valve branch).
               IF NOT "Valves_DB".Valve[#i].LocalMode AND "Valves_DB".Valve[#i].Healthy
                  AND NOT "Valves_DB".PositionFault[#i] THEN
                   // Interlock: Ignore if both commands pressed simultaneously
                   IF "Valves_DB".Valve[#i].OpenCmd AND "Valves_DB".Valve[#i].CloseCmd THEN
                       "Valves_DB".Valve[#i].OpenCmd := FALSE;
                       "Valves_DB".Valve[#i].CloseCmd := FALSE;
                   ELSIF "Valves_DB".Valve[#i].OpenCmd THEN
                       // Record the operator's intent before acting on it. Never cleared on arrival -
                       // this is what the HMI compares against actual position to spot a valve that is
                       // not where it was told to go (stuck limit switch, failed actuator).
                       "Valves_DB".CmdPos[#i] := 1;   // 1 = OPEN
                       IF "Valve_Channels_DB".OpenFbChannel[#i] > 0 THEN
                           "Valves_DB".Valve[#i].OpenValve := TRUE;
                           "Valves_DB".Valve[#i].CloseValve := FALSE;
                       ELSE
                           // Start OPENING sequence: Immediately leave seat -> MOVING!
                           "Valves_DB".Valve[#i].OpenFB := FALSE;
                           "Valves_DB".Valve[#i].ClosedFB := FALSE;
                           #SimStep[#i] := 1; // 1 = opening in progress
                       END_IF;
                       "Valves_DB".Valve[#i].OpenCmd := FALSE;
                       "Valves_DB".Valve[#i].CloseCmd := FALSE;
                   ELSIF "Valves_DB".Valve[#i].CloseCmd THEN
                       "Valves_DB".CmdPos[#i] := 2;   // 2 = CLOSE
                       IF "Valve_Channels_DB".OpenFbChannel[#i] > 0 THEN
                           "Valves_DB".Valve[#i].CloseValve := TRUE;
                           "Valves_DB".Valve[#i].OpenValve := FALSE;
                       ELSE
                           // Start CLOSING sequence: Immediately leave seat -> MOVING!
                           "Valves_DB".Valve[#i].OpenFB := FALSE;
                           "Valves_DB".Valve[#i].ClosedFB := FALSE;
                           #SimStep[#i] := 2; // 2 = closing in progress
                       END_IF;
                       "Valves_DB".Valve[#i].CloseCmd := FALSE;
                       "Valves_DB".Valve[#i].OpenCmd := FALSE;
                   END_IF;
               ELSE
                   // LOCAL MODE / UNHEALTHY: discard any pending command outright.
                   // Without this the command bit stayed latched while it was being (correctly)
                   // refused, and then executed by itself on the very next scan after the valve
                   // returned to remote/healthy - i.e. the valve moves with nobody commanding it,
                   // seconds or hours after the button was pressed. Found by live test 2026-08-15
                   // (CM79: OPEN pressed in Local, LocalMode cleared, valve immediately ran and
                   // then latched Fail-to-Open). A refused command must be forgotten, not queued.
                   "Valves_DB".Valve[#i].OpenCmd := FALSE;
                   "Valves_DB".Valve[#i].CloseCmd := FALSE;
               END_IF;

               // Real valves only: drop the run-latch the instant the real limit switch (read
               // elsewhere by FC_IoMapper) confirms arrival, and force it off on an unhealthy/local
               // transition so a stale "still running" output can't linger past a fault.
               IF "Valve_Channels_DB".OpenFbChannel[#i] > 0 THEN
                   IF "Valves_DB".Valve[#i].OpenFB THEN "Valves_DB".Valve[#i].OpenValve := FALSE; END_IF;
                   IF "Valves_DB".Valve[#i].ClosedFB THEN "Valves_DB".Valve[#i].CloseValve := FALSE; END_IF;
                   IF "Valves_DB".Valve[#i].LocalMode OR NOT "Valves_DB".Valve[#i].Healthy
                      OR "Valves_DB".PositionFault[#i] THEN
                       "Valves_DB".Valve[#i].OpenValve := FALSE;
                       "Valves_DB".Valve[#i].CloseValve := FALSE;
                   END_IF;
               END_IF;

               // 1a. Travel timeouts are self-clearing on successful arrival. A latched Fail-to-Open
               // sitting on a valve that has since opened correctly is actively misleading: the panel
               // shows FAULT on a working valve, and the operator cannot tell "broken now" from "broke
               // once, fine since". Clearing on arrival lets the alarm show raised -> cleared; it stays
               // in alarm history and still needs acknowledging, so the record survives.
               // Only the travel timeouts behave this way. UnexpMove stays latched (it is an event that
               // happened, with no natural "resolved" state) and DirFault stays latched (it points at
               // wiring, which does not fix itself and should need a deliberate human reset).
               // Note the asymmetry is deliberate: arriving OPEN clears only the open timeout. A failed
               // close leaves the valve at the open limit, so ClosedFB is false and TimeoutCloseAlarm
               // correctly survives.
               IF "Valves_DB".Valve[#i].OpenFB THEN
                   "Valves_DB".TimeoutOpenAlarm[#i] := FALSE;
               END_IF;
               IF "Valves_DB".Valve[#i].ClosedFB THEN
                   "Valves_DB".TimeoutCloseAlarm[#i] := FALSE;
               END_IF;

               // 1b. Direction / limit-switch discrepancy (H) — the physical evidence contradicts the
               // command. Driving OPEN with the CLOSED limit still made (or the mirror) after the 5s
               // grace means either the valve went the wrong way (OPEN/CLOSE swapped at the interposing
               // relays) or it never left its seat (dead actuator, stuck limit switch). The PLC cannot
               // separate those from two limit switches, and it must not try: deducing "the wiring
               // looks swapped so I will drive the other output" would bake compensation for a wiring
               // fault into safety logic, and every valve would invert the day someone fixed the wiring.
               // So: stop driving, latch, and let a human look at it.
               // The IN condition self-resets the timer the moment the contradiction clears, so a
               // normal stroke leaving its seat within the grace never arms this.
               "Valves_DB".DirTmr[#i](
                   IN := ("Valves_DB".Valve[#i].OpenValve AND "Valves_DB".Valve[#i].ClosedFB)
                         OR ("Valves_DB".Valve[#i].CloseValve AND "Valves_DB".Valve[#i].OpenFB),
                   PT := #seatPT);
               IF "Valves_DB".DirTmr[#i].Q THEN
                   "Valves_DB".DirFault[#i] := TRUE;
                   // Fail safe: when direction is in doubt, stop. Continuing to energise would keep
                   // opening a valve somebody asked to close.
                   "Valves_DB".Valve[#i].OpenValve := FALSE;
                   "Valves_DB".Valve[#i].CloseValve := FALSE;
               END_IF;

               // 2. Motion Delay Execution — real 3.0s TON per valve (Valve[i].TimerOpen/Close
               // are dedicated instances since they live inside this array element). Scan-cycle
               // counting was used before; it only equalled 3.0s if every scan took exactly
               // 100ms, which isn't guaranteed, so the MOVING state could flash by in well
               // under a second on a fast scan. A TON runs on the CPU's real-time clock, so
               // this duration is exact regardless of scan speed.
               // Stuck (set via the popup's SIMULATE STUCK toggle) holds the valve at the normal
               // 3s completion so it never arrives — TON.ET keeps counting past PT as long as IN
               // stays true, so at 8s (well past the normal 3s travel) that's a genuine failure to
               // arrive, not just "still moving": latch Fail to Open/Close (C/D) and give up on the
               // sequence, leaving both feedbacks false (position genuinely unknown).
               // IN covers both cases: SimStep=1 during a simulated open travel, OpenValve latched
               // true during a real one - the two are mutually exclusive per valve (Section 1 only
               // ever sets one or the other for a given i), so sharing the one TON instance is safe.
               "Valves_DB".Valve[#i].TimerOpen(IN := (#SimStep[#i] = 1) OR "Valves_DB".Valve[#i].OpenValve, PT := #travelPT);
               IF #SimStep[#i] = 1 THEN
                   IF NOT "Valves_DB".Stuck[#i] AND "Valves_DB".Valve[#i].TimerOpen.ET >= T#3S THEN
                       "Valves_DB".Valve[#i].OpenFB := TRUE;   // Reached OPEN position!
                       "Valves_DB".Valve[#i].ClosedFB := FALSE;
                       #SimStep[#i] := 0;                       // Sequence complete
                   ELSIF "Valves_DB".Valve[#i].TimerOpen.Q THEN
                       "Valves_DB".TimeoutOpenAlarm[#i] := TRUE;  // Fail to Open (C)
                       "Valves_DB".Valve[#i].OpenFB := FALSE;
                       "Valves_DB".Valve[#i].ClosedFB := FALSE;
                       #SimStep[#i] := 0;
                   END_IF;
               ELSIF "Valves_DB".Valve[#i].OpenValve AND "Valves_DB".Valve[#i].TimerOpen.Q THEN
                   // Real valve commanded open 8s ago and the real limit switch never confirmed -
                   // genuine failure to open. Give up on the run output; position stays whatever the
                   // real feedback says (already false, or this wouldn't still be latched).
                   "Valves_DB".TimeoutOpenAlarm[#i] := TRUE;  // Fail to Open (C)
                   "Valves_DB".Valve[#i].OpenValve := FALSE;
               END_IF;

               "Valves_DB".Valve[#i].TimerClose(IN := (#SimStep[#i] = 2) OR "Valves_DB".Valve[#i].CloseValve, PT := #travelPT);
               IF #SimStep[#i] = 2 THEN
                   IF NOT "Valves_DB".Stuck[#i] AND "Valves_DB".Valve[#i].TimerClose.ET >= T#3S THEN
                       "Valves_DB".Valve[#i].ClosedFB := TRUE; // Reached CLOSED position!
                       "Valves_DB".Valve[#i].OpenFB := FALSE;
                       #SimStep[#i] := 0;                       // Sequence complete
                   ELSIF "Valves_DB".Valve[#i].TimerClose.Q THEN
                       "Valves_DB".TimeoutCloseAlarm[#i] := TRUE; // Fail to Close (D)
                       "Valves_DB".Valve[#i].OpenFB := FALSE;
                       "Valves_DB".Valve[#i].ClosedFB := FALSE;
                       #SimStep[#i] := 0;
                   END_IF;
               ELSIF "Valves_DB".Valve[#i].CloseValve AND "Valves_DB".Valve[#i].TimerClose.Q THEN
                   "Valves_DB".TimeoutCloseAlarm[#i] := TRUE; // Fail to Close (D)
                   "Valves_DB".Valve[#i].CloseValve := FALSE;
               END_IF;

               // 3. Failsafe Double Indication Fault Check
               // Both limit switches made at once is physically impossible - a wiring or
               // sensor fault. This used to force Healthy := FALSE, but Healthy is a
               // VALVE-OWNED signal: the actuator's own health contact. Overwriting it with
               // our conclusion meant one event raised BOTH _DoubleInd and _Unhealthy, and
               // the second ("CMxx reported Unhealthy status") was false - it sent a
               // technician to the actuator when the fault is in the limit switches.
               // Split into its own flag 2026-09-06 (item 12). Healthy is now read-only
               // everywhere; FC_IoMapper's raw DI read is its only writer in the program.
               // Plain assignment, NOT a latch: the condition is either physically present
               // or it is not, and it must clear itself when the limits stop conflicting.
               "Valves_DB".PositionFault[#i] := "Valves_DB".Valve[#i].OpenFB AND "Valves_DB".Valve[#i].ClosedFB;

               // 3a. Alarm conditions E (Loss of Position) and F (Unexpected Movement) — both
               // derived from the exact same OpenFB/ClosedFB pair used everywhere else; the only
               // extra ingredient is TIME and CONTEXT (was a command active, what did it say a
               // moment ago), not any new signal.
               //
               // E: idle (SimStep=0, so no travel is legitimately in progress) with NEITHER limit
               // switch made — held for 2s via PosLostTmr so a normal in-flight transition can't
               // false-trip it. Suppressed while a timeout (C/D) is already latched, since that is
               // the exact same physical symptom (no position) already alarmed under its own name.
               // NOT OpenValve/CloseValve added so a real valve mid-travel (both feedbacks
               // legitimately false while the run output is latched) doesn't false-trip this the
               // same way SimStep=0 already excludes a simulated valve mid-travel.
               "Valves_DB".PosLostTmr[#i](
                   IN := (#SimStep[#i] = 0) AND NOT "Valves_DB".Valve[#i].OpenValve
                         AND NOT "Valves_DB".Valve[#i].CloseValve
                         AND NOT "Valves_DB".Valve[#i].OpenFB
                         AND NOT "Valves_DB".Valve[#i].ClosedFB
                         AND NOT "Valves_DB".TimeoutOpenAlarm[#i] AND NOT "Valves_DB".TimeoutCloseAlarm[#i],
                   PT := T#2S);

               // F: a limit switch that WAS made a scan ago has dropped, with no travel sequence
               // running to explain it — nobody commanded this, so something moved the valve
               // (handwheel) or a switch/wiring fault occurred. Latched.
               // Requires SimStep to have been 0 BOTH before and after this scan's processing: a
               // fresh command (0 -> nonzero, in section 1) or a completing travel (nonzero -> 0,
               // in section 2) each only satisfy ONE side of this, so both are correctly excluded —
               // only a scan truly idle throughout can reach here.
               // Real valves: also require the run-latch off both before and after, same reasoning
               // as SimStep above - a real valve leaving its seat on a legitimate command is not
               // "unexplained" just because OpenValve/CloseValve doesn't happen to be SimStep.
               IF #simStepAtStart = 0 AND #SimStep[#i] = 0
                  AND NOT "Valves_DB".Valve[#i].OpenValve AND NOT "Valves_DB".Valve[#i].CloseValve THEN
                   IF ("Valves_DB".PrevOpenFB[#i] AND NOT "Valves_DB".Valve[#i].OpenFB) OR
                      ("Valves_DB".PrevClosedFB[#i] AND NOT "Valves_DB".Valve[#i].ClosedFB) THEN
                       "Valves_DB".UnexpMove[#i] := TRUE;
                   END_IF;
               END_IF;
               "Valves_DB".PrevOpenFB[#i] := "Valves_DB".Valve[#i].OpenFB;
               "Valves_DB".PrevClosedFB[#i] := "Valves_DB".Valve[#i].ClosedFB;

               // 4. Priority Summary Counting — plant-wide AND per-zone in the same pass
               // (this loop already runs 1..89 every scan regardless, so the zone-scoped
               // increments below are free — they're what let every HMI KPI/caption cell
               // read one tag instead of re-looping its zone's 28-32 valves itself).
               // Zone valve-number ranges follow physical position from stern to bow, so the HMI
               // mimic reads slots straight across: AFT=1-27, ER=28-54, FWD=55-89. Exact fit to the
               // client schedule's real 27/27/35 = 89 valves - no spare padding slots anywhere.
               #tempConfigured := #tempConfigured + 1;
               IF #i <= 27 THEN
                   #tempAftConfigured := #tempAftConfigured + 1;
               ELSIF #i <= 54 THEN
                   #tempErConfigured := #tempErConfigured + 1;
               ELSE
                   #tempFwdConfigured := #tempFwdConfigured + 1;
               END_IF;

               // StateCode is assigned in these same branches (0=UNCONFIGURED 1=FAULT 2=LOCAL
               // 3=OPEN 4=CLOSED 5=MOVING) so the HMI reads one Int per valve instead of
               // recombining five raw bits in JavaScript on every refresh.
               // UnexpMove (F) and PosLostTmr.Q (E) added here so a valve with a genuine position
               // problem shows FAULT instead of falling through to the default MOVING bucket below,
               // which was otherwise indistinguishable from a normal in-flight transition - the exact
               // blind spot E was designed to close, but the display logic was never updated to match.
               // Position-only code — the same chain as StateCode below but WITHOUT the fault branch,
               // so a faulted valve still reports where it is. The popup shows this alongside the
               // fault rather than instead of it.
               IF "Valves_DB".Valve[#i].OpenValve THEN
                   "Valves_DB".PosCode[#i] := 6;
               ELSIF "Valves_DB".Valve[#i].CloseValve THEN
                   "Valves_DB".PosCode[#i] := 7;
               ELSIF "Valves_DB".Valve[#i].OpenFB AND NOT "Valves_DB".Valve[#i].ClosedFB THEN
                   "Valves_DB".PosCode[#i] := 3;
               ELSIF NOT "Valves_DB".Valve[#i].OpenFB AND "Valves_DB".Valve[#i].ClosedFB THEN
                   "Valves_DB".PosCode[#i] := 4;
               ELSE
                   "Valves_DB".PosCode[#i] := 5;
               END_IF;

               // Fault reason, most specific first. Double indication is tested before Healthy because
               // it is what FORCES Healthy false — checking Healthy first would mask the real cause
               // behind a generic "unhealthy".
               IF "Valves_DB".PositionFault[#i] THEN
                   "Valves_DB".FaultCode[#i] := 2;
               ELSIF "Valves_DB".DirFault[#i] THEN
                   "Valves_DB".FaultCode[#i] := 7;
               ELSIF "Valves_DB".TimeoutOpenAlarm[#i] THEN
                   "Valves_DB".FaultCode[#i] := 3;
               ELSIF "Valves_DB".TimeoutCloseAlarm[#i] THEN
                   "Valves_DB".FaultCode[#i] := 4;
               ELSIF "Valves_DB".UnexpMove[#i] THEN
                   "Valves_DB".FaultCode[#i] := 6;
               ELSIF "Valves_DB".PosLostTmr[#i].Q THEN
                   "Valves_DB".FaultCode[#i] := 5;
               ELSIF NOT "Valves_DB".Valve[#i].Healthy THEN
                   "Valves_DB".FaultCode[#i] := 1;
               ELSE
                   "Valves_DB".FaultCode[#i] := 0;
               END_IF;

               // What the mimic box should show right now, flashing included. Computing the
               // ALTERNATION here means the HMI binds one native value map and runs no scripts at all
               // - 89 scripted boxes re-evaluating on every clock tick would be real load on the panel,
               // and this project already learned that lesson with the popup.
               // When nothing is faulted DispCode simply equals PosCode and never changes, so a healthy
               // plant produces zero tag traffic. Cost scales with faults, not with valve count.
               IF NOT "Valves_DB".Valve[#i].Configured THEN
                   "Valves_DB".DispCode[#i] := 0;
               ELSIF "Valves_DB".FaultCode[#i] > 0 AND "Valves_DB".Clock_Flash THEN
                   "Valves_DB".DispCode[#i] := 1;                                  // red half of the flash
               ELSIF "Valves_DB".Valve[#i].LocalMode THEN
                   "Valves_DB".DispCode[#i] := 2;                                  // amber, steady
               ELSE
                   "Valves_DB".DispCode[#i] := "Valves_DB".PosCode[#i];        // position
               END_IF;

